C05487=1118.732,158.119,-61.971,-179.423,8.843,149.556
C05488=1118.727,158.349,-61.992,-179.422,8.846,149.556
C05489=1118.724,158.578,-62.012,-179.419,8.849,149.556
C05490=1118.719,158.807,-62.033,-179.417,8.852,149.556
C05491=1118.714,159.056,-62.056,-179.415,8.856,149.557
C05492=1118.710,159.305,-62.078,-179.412,8.859,149.557
C05493=1118.706,159.554,-62.100,-179.410,8.862,149.557
C05494=1118.701,159.803,-62.123,-179.408,8.865,149.557
C05495=1118.696,160.052,-62.145,-179.406,8.869,149.557
C05496=1118.691,160.301,-62.168,-179.403,8.872,149.557
C05497=1118.687,160.550,-62.191,-179.401,8.875,149.558
C05498=1118.683,160.799,-62.213,-179.399,8.878,149.558
C05499=1118.677,161.048,-62.236,-179.397,8.881,149.558
C05500=1118.674,161.296,-62.259,-179.394,8.884,149.558
C05501=1118.668,161.546,-62.281,-179.392,8.887,149.558
C05502=1118.664,161.794,-62.304,-179.390,8.891,149.558
C05503=1118.659,162.044,-62.326,-179.387,8.894,149.558
C05504=1118.655,162.292,-62.349,-179.385,8.898,149.558
C05505=1118.650,162.542,-62.372,-179.383,8.901,149.558
C05506=1118.645,162.790,-62.394,-179.380,8.904,149.558
C05507=1118.641,163.039,-62.417,-179.378,8.907,149.559
C05508=1118.636,163.288,-62.440,-179.376,8.910,149.559
C05509=1118.632,163.537,-62.463,-179.373,8.914,149.559
C05510=1118.627,163.785,-62.485,-179.372,8.916,149.559
C05511=1118.622,164.035,-62.508,-179.369,8.919,149.559
C05512=1118.618,164.284,-62.531,-179.367,8.923,149.559
C05513=1118.614,164.533,-62.554,-179.364,8.926,149.559
C05514=1118.609,164.781,-62.576,-179.362,8.929,149.559
C05515=1118.604,165.031,-62.599,-179.360,8.932,149.560
C05516=1118.600,165.279,-62.622,-179.357,8.936,149.560
C05517=1118.595,165.528,-62.645,-179.355,8.939,149.560
C05518=1118.591,165.777,-62.669,-179.353,8.941,149.560
C05519=1118.586,166.026,-62.690,-179.351,8.945,149.560
C05520=1118.581,166.275,-62.714,-179.348,8.948,149.560
C05521=1118.576,166.524,-62.737,-179.346,8.951,149.560
C05522=1118.572,166.773,-62.760,-179.344,8.954,149.560
C05523=1118.568,167.022,-62.783,-179.341,8.957,149.560
C05524=1118.562,167.271,-62.805,-179.340,8.960,149.560
C05525=1118.558,167.519,-62.828,-179.337,8.963,149.560
C05526=1118.553,167.768,-62.852,-179.335,8.966,149.561
C05527=1118.549,168.017,-62.875,-179.333,8.970,149.561
C05528=1118.545,168.266,-62.898,-179.330,8.973,149.561
C05529=1118.540,168.515,-62.921,-179.328,8.975,149.561
C05530=1118.535,168.764,-62.944,-179.326,8.979,149.561
C05531=1118.531,169.012,-62.967,-179.324,8.982,149.561
C05532=1118.526,169.261,-62.990,-179.321,8.985,149.561
C05533=1118.521,169.510,-63.013,-179.320,8.988,149.561
C05534=1118.517,169.759,-63.037,-179.317,8.991,149.561
C05535=1118.512,170.009,-63.059,-179.315,8.994,149.561
C05536=1118.508,170.258,-63.082,-179.312,8.997,149.561
C05537=1118.503,170.507,-63.106,-179.311,9.000,149.562
C05538=1118.498,170.755,-63.129,-179.308,9.003,149.562
C05539=1118.494,170.969,-63.149,-179.306,9.005,149.562
C05540=1118.491,171.183,-63.169,-179.304,9.009,149.562
C05541=1118.487,171.397,-63.188,-179.302,9.011,149.562
C05542=1118.482,171.610,-63.209,-179.300,9.013,149.562
C05543=1118.479,171.824,-63.229,-179.298,9.016,149.562
C05544=1118.475,172.038,-63.248,-179.297,9.018,149.562
C05545=1118.471,172.252,-63.269,-179.294,9.021,149.562
C05546=1118.467,172.466,-63.289,-179.292,9.024,149.562
C05547=1118.462,172.715,-63.312,-179.291,9.026,149.562
C05548=1118.458,172.964,-63.336,-179.289,9.029,149.563
C05549=1118.453,173.213,-63.359,-179.286,9.033,149.563
C05550=1118.449,173.461,-63.382,-179.283,9.036,149.563
C05551=1118.444,173.710,-63.405,-179.282,9.038,149.563
C05552=1118.439,173.958,-63.429,-179.279,9.042,149.563
C05553=1118.435,174.207,-63.452,-179.277,9.045,149.563
C05554=1118.430,174.456,-63.476,-179.275,9.047,149.563
C05555=1118.425,174.705,-63.499,-179.273,9.050,149.563
C05556=1118.421,174.954,-63.522,-179.270,9.054,149.563
C05557=1118.416,175.203,-63.546,-179.269,9.056,149.564
C05558=1118.412,175.451,-63.569,-179.266,9.059,149.564
C05559=1118.408,175.701,-63.592,-179.264,9.062,149.564
C05560=1118.403,175.950,-63.616,-179.262,9.065,149.564
C05561=1118.398,176.198,-63.640,-179.260,9.068,149.564
C05562=1118.394,176.447,-63.663,-179.257,9.071,149.564
C05563=1118.389,176.696,-63.687,-179.256,9.074,149.564
C05564=1118.385,176.944,-63.711,-179.253,9.077,149.564
C05565=1118.380,177.193,-63.734,-179.251,9.080,149.564
C05566=1118.375,177.442,-63.757,-179.249,9.083,149.564
C05567=1118.371,177.692,-63.782,-179.247,9.086,149.565
C05568=1118.367,177.941,-63.805,-179.244,9.089,149.565
C05569=1118.362,178.190,-63.829,-179.243,9.092,149.565
C05570=1118.358,178.438,-63.853,-179.240,9.095,149.565
C05571=1118.353,178.687,-63.876,-179.239,9.097,149.565
C05572=1118.348,178.936,-63.899,-179.236,9.100,149.565
C05573=1118.344,179.185,-63.923,-179.234,9.104,149.565
C05574=1118.339,179.434,-63.947,-179.231,9.107,149.565
C05575=1118.335,179.682,-63.971,-179.229,9.110,149.565
C05576=1118.330,179.931,-63.994,-179.226,9.113,149.565
C05577=1118.326,180.179,-64.018,-179.224,9.116,149.565
C05578=1118.321,180.428,-64.042,-179.221,9.120,149.565
C05579=1118.317,180.677,-64.066,-179.219,9.123,149.566
C05580=1118.313,180.927,-64.089,-179.215,9.126,149.565
C05581=1118.308,181.175,-64.114,-179.213,9.129,149.565
C05582=1118.303,181.424,-64.137,-179.210,9.132,149.565
C05583=1118.298,181.673,-64.162,-179.208,9.135,149.566
C05584=1118.294,181.922,-64.185,-179.205,9.139,149.566
C05585=1118.289,182.170,-64.209,-179.203,9.142,149.566
C05586=1118.285,182.419,-64.232,-179.200,9.145,149.566
C05587=1118.281,182.668,-64.257,-179.198,9.148,149.566
C05588=1118.276,182.917,-64.281,-179.195,9.151,149.566
C05589=1118.272,183.166,-64.304,-179.192,9.154,149.566
C05590=1118.266,183.415,-64.329,-179.190,9.157,149.566
C05591=1118.262,183.663,-64.353,-179.187,9.160,149.566
C05592=1118.257,183.912,-64.376,-179.184,9.163,149.566
C05593=1118.254,184.161,-64.401,-179.183,9.165,149.566
C05594=1118.249,184.410,-64.425,-179.180,9.169,149.566
C05595=1118.245,184.623,-64.445,-179.178,9.172,149.566
C05596=1118.240,184.837,-64.466,-179.176,9.174,149.566
C05597=1118.237,185.051,-64.487,-179.174,9.176,149.566
C05598=1118.233,185.264,-64.508,-179.172,9.179,149.566
C05599=1118.229,185.479,-64.528,-179.169,9.182,149.566
C05600=1118.226,185.692,-64.549,-179.167,9.184,149.566
C05601=1118.221,185.906,-64.569,-179.165,9.186,149.566
C05602=1118.218,186.120,-64.591,-179.163,9.188,149.566
C05603=1118.213,186.369,-64.614,-179.161,9.191,149.566
C05604=1118.208,186.617,-64.638,-179.158,9.195,149.566
C05605=1118.203,186.866,-64.663,-179.156,9.198,149.566
C05606=1118.200,187.115,-64.687,-179.154,9.200,149.566
C05607=1118.195,187.363,-64.711,-179.151,9.203,149.566
C05608=1118.190,187.612,-64.736,-179.149,9.206,149.566
C05609=1118.185,187.861,-64.759,-179.147,9.209,149.566
C05610=1118.182,188.110,-64.784,-179.144,9.212,149.566
C05611=1118.176,188.359,-64.809,-179.142,9.215,149.566
C05612=1118.172,188.607,-64.833,-179.140,9.217,149.566
C05613=1118.168,188.856,-64.857,-179.137,9.220,149.566
C05614=1118.163,189.105,-64.882,-179.135,9.223,149.566
C05615=1118.159,189.353,-64.906,-179.133,9.226,149.566
C05616=1118.154,189.602,-64.930,-179.130,9.229,149.566
C05617=1118.149,189.851,-64.955,-179.129,9.231,149.567
C05618=1118.145,190.100,-64.979,-179.126,9.234,149.567
C05619=1118.140,190.348,-65.004,-179.124,9.237,149.567
C05620=1118.136,190.597,-65.028,-179.122,9.240,149.567
C05621=1118.132,190.846,-65.052,-179.120,9.242,149.567
C05622=1118.127,191.095,-65.077,-179.117,9.245,149.567
C05623=1118.123,191.343,-65.101,-179.115,9.247,149.567
C05624=1118.118,191.593,-65.126,-179.114,9.250,149.567
C05625=1118.114,191.841,-65.150,-179.111,9.253,149.567
C05626=1118.108,192.090,-65.175,-179.109,9.256,149.567
C05627=1118.105,192.339,-65.199,-179.107,9.259,149.567
C05628=1118.100,192.588,-65.224,-179.105,9.261,149.567
C05629=1118.095,192.836,-65.248,-179.103,9.264,149.567
C05630=1118.091,193.085,-65.273,-179.101,9.267,149.567
C05631=1118.086,193.334,-65.297,-179.099,9.269,149.568
C05632=1118.082,193.582,-65.321,-179.097,9.272,149.568
C05633=1118.077,193.832,-65.346,-179.095,9.275,149.568
C05634=1118.073,194.079,-65.371,-179.093,9.277,149.568
C05635=1118.069,194.329,-65.396,-179.091,9.280,149.568
C05636=1118.064,194.578,-65.421,-179.089,9.283,149.568
C05637=1118.059,194.826,-65.445,-179.087,9.285,149.568
C05638=1118.055,195.075,-65.470,-179.085,9.289,149.568
C05639=1118.050,195.324,-65.494,-179.083,9.291,149.568
C05640=1118.045,195.572,-65.519,-179.081,9.294,149.568
C05641=1118.042,195.821,-65.544,-179.080,9.296,149.569
C05642=1118.037,196.070,-65.568,-179.077,9.299,149.569
C05643=1118.033,196.319,-65.593,-179.076,9.302,149.569
C05644=1118.028,196.567,-65.618,-179.073,9.305,149.569
C05645=1118.023,196.816,-65.643,-179.070,9.309,149.569
C05646=1118.019,197.065,-65.667,-179.067,9.313,149.569
C05647=1118.014,197.314,-65.692,-179.064,9.315,149.569
C05648=1118.010,197.562,-65.717,-179.061,9.319,149.569
C05649=1118.005,197.811,-65.742,-179.058,9.322,149.569
C05650=1118.001,198.060,-65.767,-179.054,9.325,149.569
C05651=1117.996,198.273,-65.788,-179.052,9.329,149.569
C05652=1117.993,198.487,-65.809,-179.049,9.331,149.569
C05653=1117.989,198.700,-65.831,-179.047,9.334,149.569
C05654=1117.985,198.914,-65.853,-179.044,9.336,149.568
C05655=1117.982,199.128,-65.874,-179.041,9.339,149.568
C05656=1117.978,199.341,-65.895,-179.038,9.342,149.568
C05657=1117.974,199.555,-65.917,-179.036,9.345,149.568
C05658=1117.970,199.768,-65.938,-179.033,9.347,149.568
C05659=1117.965,200.017,-65.964,-179.030,9.351,149.568
C05660=1117.961,200.266,-65.988,-179.027,9.354,149.568
C05661=1117.957,200.514,-66.013,-179.024,9.357,149.568
C05662=1117.952,200.763,-66.038,-179.021,9.360,149.568
C05663=1117.948,201.012,-66.063,-179.018,9.363,149.568
C05664=1117.944,201.261,-66.088,-179.015,9.366,149.568
C05665=1117.939,201.509,-66.114,-179.012,9.369,149.568
C05666=1117.934,201.759,-66.139,-179.009,9.372,149.567
C05667=1117.930,202.006,-66.163,-179.006,9.375,149.568
C05668=1117.926,202.256,-66.189,-179.003,9.378,149.567
C05669=1117.921,202.504,-66.214,-179.000,9.381,149.567
C05670=1117.917,202.753,-66.240,-178.997,9.384,149.567
C05671=1117.912,203.002,-66.265,-178.994,9.388,149.567
C05672=1117.907,203.250,-66.290,-178.991,9.390,149.567
C05673=1117.904,203.499,-66.315,-178.988,9.393,149.567
C05674=1117.899,203.747,-66.340,-178.985,9.396,149.567
C05675=1117.895,203.996,-66.366,-178.982,9.398,149.567
C05676=1117.890,204.244,-66.391,-178.980,9.402,149.567
C05677=1117.885,204.494,-66.416,-178.977,9.404,149.566
C05678=1117.881,204.743,-66.442,-178.973,9.408,149.566
C05679=1117.876,204.991,-66.467,-178.970,9.411,149.566
C05680=1117.872,205.240,-66.492,-178.968,9.414,149.566
C05681=1117.867,205.489,-66.518,-178.965,9.416,149.566
C05682=1117.863,205.737,-66.543,-178.962,9.419,149.566
C05683=1117.859,205.985,-66.569,-178.959,9.422,149.566
C05684=1117.854,206.234,-66.594,-178.957,9.425,149.566
C05685=1117.850,206.483,-66.619,-178.954,9.428,149.566
C05686=1117.845,206.732,-66.645,-178.951,9.431,149.566
C05687=1117.841,206.980,-66.670,-178.948,9.434,149.566
C05688=1117.836,207.229,-66.696,-178.945,9.436,149.566
C05689=1117.832,207.478,-66.722,-178.942,9.439,149.565
C05690=1117.827,207.726,-66.747,-178.940,9.442,149.565
C05691=1117.823,207.974,-66.773,-178.937,9.445,149.565
C05692=1117.819,208.223,-66.798,-178.934,9.448,149.565
C05693=1117.814,208.471,-66.824,-178.932,9.450,149.565
C05694=1117.810,208.721,-66.849,-178.929,9.453,149.565
C05695=1117.805,208.970,-66.875,-178.926,9.456,149.565
C05696=1117.800,209.219,-66.901,-178.924,9.459,149.565
C05697=1117.796,209.467,-66.926,-178.921,9.462,149.565
C05698=1117.791,209.716,-66.952,-178.918,9.465,149.565
C05699=1117.787,209.964,-66.978,-178.915,9.468,149.565
C05700=1117.783,210.213,-67.004,-178.913,9.471,149.565
C05701=1117.778,210.461,-67.029,-178.910,9.473,149.565
C05702=1117.774,210.710,-67.055,-178.907,9.477,149.565
C05703=1117.770,210.958,-67.081,-178.906,9.479,149.565
C05704=1117.766,211.207,-67.107,-178.903,9.482,149.565
C05705=1117.761,211.455,-67.132,-178.900,9.485,149.565
C05706=1117.756,211.704,-67.159,-178.898,9.488,149.565
C05707=1117.753,211.918,-67.181,-178.896,9.490,149.565
C05708=1117.749,212.132,-67.202,-178.893,9.493,149.565
C05709=1117.744,212.345,-67.225,-178.891,9.496,149.565
C05710=1117.741,212.558,-67.247,-178.889,9.498,149.565
C05711=1117.737,212.772,-67.270,-178.887,9.501,149.565
C05712=1117.733,212.985,-67.291,-178.885,9.503,149.565
C05713=1117.729,213.199,-67.314,-178.883,9.506,149.565
C05714=1117.726,213.412,-67.336,-178.881,9.508,149.565
C05715=1117.721,213.661,-67.362,-178.879,9.511,149.565
C05716=1117.717,213.909,-67.387,-178.877,9.514,149.565
C05717=1117.712,214.158,-67.414,-178.875,9.517,149.566
C05718=1117.708,214.407,-67.440,-178.873,9.519,149.566
C05719=1117.704,214.655,-67.466,-178.870,9.522,149.566
C05720=1117.700,214.904,-67.492,-178.868,9.525,149.566
C05721=1117.694,215.152,-67.518,-178.866,9.528,149.566
C05722=1117.690,215.401,-67.544,-178.864,9.531,149.566
C05723=1117.686,215.650,-67.570,-178.862,9.534,149.566
C05724=1117.682,215.898,-67.596,-178.860,9.537,149.566
C05725=1117.677,216.147,-67.623,-178.858,9.539,149.567
C05726=1117.673,216.396,-67.648,-178.855,9.543,149.567
C05727=1117.669,216.645,-67.674,-178.853,9.546,149.567
C05728=1117.664,216.892,-67.700,-178.851,9.548,149.567
C05729=1117.659,217.141,-67.727,-178.849,9.552,149.567
C05730=1117.655,217.389,-67.753,-178.846,9.555,149.567
C05731=1117.651,217.638,-67.779,-178.844,9.558,149.567
C05732=1117.646,217.887,-67.805,-178.842,9.560,149.567
C05733=1117.642,218.135,-67.832,-178.840,9.564,149.567
C05734=1117.638,218.384,-67.857,-178.837,9.567,149.567
C05735=1117.633,218.633,-67.884,-178.835,9.570,149.568
C05736=1117.629,218.882,-67.910,-178.833,9.573,149.568
C05737=1117.625,219.130,-67.936,-178.831,9.576,149.568
C05738=1117.620,219.378,-67.963,-178.828,9.579,149.568
C05739=1117.615,219.627,-67.988,-178.826,9.582,149.568
C05740=1117.611,219.875,-68.015,-178.824,9.585,149.568
C05741=1117.606,220.124,-68.041,-178.821,9.588,149.568
C05742=1117.602,220.372,-68.068,-178.818,9.591,149.568
C05743=1117.598,220.622,-68.094,-178.816,9.595,149.568
C05744=1117.594,220.870,-68.121,-178.813,9.598,149.569
C05745=1117.589,221.118,-68.148,-178.811,9.601,149.569
C05746=1117.585,221.367,-68.173,-178.808,9.604,149.569
C05747=1117.581,221.615,-68.200,-178.806,9.607,149.569
C05748=1117.576,221.864,-68.226,-178.803,9.610,149.569
C05749=1117.572,222.113,-68.253,-178.801,9.613,149.569
C05750=1117.567,222.361,-68.280,-178.798,9.616,149.569
C05751=1117.563,222.610,-68.305,-178.796,9.619,149.569
C05752=1117.558,222.858,-68.332,-178.793,9.623,149.569
C05753=1117.554,223.107,-68.358,-178.791,9.626,149.569
C05754=1117.550,223.356,-68.385,-178.788,9.629,149.569
C05755=1117.546,223.604,-68.412,-178.786,9.632,149.569
C05756=1117.541,223.852,-68.439,-178.783,9.635,149.569
C05757=1117.537,224.101,-68.465,-178.781,9.638,149.569
C05758=1117.532,224.350,-68.492,-178.778,9.641,149.569
C05759=1117.527,224.598,-68.519,-178.774,9.645,149.569
C05760=1117.523,224.846,-68.545,-178.772,9.648,149.569
C05761=1117.519,225.095,-68.572,-178.769,9.651,149.569
C05762=1117.515,225.344,-68.598,-178.767,9.654,149.570
C05763=1117.511,225.557,-68.621,-178.764,9.657,149.570
C05764=1117.507,225.770,-68.644,-178.762,9.659,149.569
C05765=1117.503,225.984,-68.667,-178.759,9.662,149.570
C05766=1117.500,226.197,-68.690,-178.757,9.665,149.570
C05767=1117.496,226.410,-68.713,-178.755,9.667,149.569
C05768=1117.492,226.624,-68.736,-178.752,9.670,149.570
C05769=1117.488,226.837,-68.759,-178.750,9.674,149.570
C05770=1117.484,227.051,-68.782,-178.747,9.676,149.569
C05771=1117.480,227.299,-68.808,-178.744,9.679,149.570
C05772=1117.476,227.548,-68.836,-178.741,9.682,149.569
C05773=1117.471,227.796,-68.863,-178.739,9.685,149.569
C05774=1117.467,228.045,-68.889,-178.736,9.688,149.569
C05775=1117.463,228.293,-68.916,-178.733,9.692,149.569
C05776=1117.458,228.542,-68.943,-178.730,9.695,149.569
C05777=1117.453,228.790,-68.970,-178.727,9.697,149.569
C05778=1117.449,229.038,-68.997,-178.723,9.701,149.569
C05779=1117.445,229.287,-69.024,-178.721,9.704,149.569
C05780=1117.441,229.536,-69.051,-178.717,9.708,149.569
C05781=1117.437,229.784,-69.078,-178.714,9.711,149.569
C05782=1117.432,230.033,-69.105,-178.711,9.713,149.569
C05783=1117.428,230.281,-69.132,-178.708,9.717,149.569
C05784=1117.423,230.530,-69.159,-178.705,9.720,149.569
C05785=1117.418,230.778,-69.186,-178.702,9.722,149.569
C05786=1117.415,231.027,-69.213,-178.698,9.726,149.568
C05787=1117.410,231.276,-69.240,-178.695,9.729,149.568
C05788=1117.406,231.523,-69.268,-178.693,9.732,149.568
C05789=1117.401,231.772,-69.295,-178.690,9.735,149.568
C05790=1117.397,232.020,-69.322,-178.687,9.737,149.568
C05791=1117.393,232.270,-69.349,-178.683,9.741,149.568
C05792=1117.389,232.518,-69.376,-178.681,9.744,149.568
C05793=1117.384,232.766,-69.404,-178.678,9.746,149.568
C05794=1117.380,233.014,-69.431,-178.675,9.749,149.568
C05795=1117.375,233.263,-69.458,-178.672,9.752,149.568
C05796=1117.371,233.512,-69.485,-178.669,9.755,149.568
C05797=1117.367,233.760,-69.513,-178.666,9.758,149.567
C05798=1117.362,234.008,-69.540,-178.663,9.760,149.567
C05799=1117.358,234.257,-69.567,-178.660,9.763,149.567
C05800=1117.353,234.506,-69.594,-178.657,9.766,149.567
C05801=1117.350,234.754,-69.622,-178.654,9.769,149.567
C05802=1117.345,235.002,-69.649,-178.652,9.771,149.567
C05803=1117.341,235.251,-69.677,-178.649,9.775,149.567
C05804=1117.337,235.499,-69.704,-178.647,9.777,149.567
C05805=1117.332,235.748,-69.731,-178.644,9.779,149.567
C05806=1117.327,235.995,-69.759,-178.641,9.782,149.567
C05807=1117.323,236.245,-69.786,-178.638,9.785,149.566
C05808=1117.319,236.493,-69.813,-178.635,9.788,149.566
C05809=1117.314,236.741,-69.841,-178.633,9.789,149.566
C05810=1117.310,236.990,-69.868,-178.630,9.793,149.566
C05811=1117.306,237.238,-69.896,-178.627,9.795,149.566
C05812=1117.301,237.487,-69.923,-178.624,9.798,149.566
C05813=1117.298,237.735,-69.951,-178.622,9.800,149.566
C05814=1117.293,237.984,-69.978,-178.619,9.803,149.566
C05815=1117.289,238.232,-70.006,-178.616,9.806,149.566
C05816=1117.284,238.481,-70.034,-178.614,9.808,149.566
C05817=1117.279,238.729,-70.062,-178.611,9.811,149.566
C05818=1117.275,238.977,-70.089,-178.609,9.813,149.566
C05819=1117.272,239.191,-70.113,-178.606,9.816,149.565
C05820=1117.268,239.404,-70.137,-178.604,9.818,149.565
C05821=1117.264,239.617,-70.160,-178.602,9.820,149.565
C05822=1117.261,239.830,-70.184,-178.600,9.822,149.565
C05823=1117.257,240.044,-70.209,-178.598,9.824,149.565
C05824=1117.253,240.257,-70.232,-178.596,9.826,149.565
C05825=1117.249,240.470,-70.256,-178.594,9.829,149.565
C05826=1117.246,240.683,-70.279,-178.591,9.831,149.565
C05827=1117.242,240.931,-70.307,-178.589,9.833,149.565
C05828=1117.237,241.180,-70.335,-178.586,9.836,149.565
C05829=1117.233,241.429,-70.363,-178.584,9.838,149.565
C05830=1117.228,241.677,-70.391,-178.582,9.841,149.565
C05831=1117.224,241.926,-70.418,-178.579,9.843,149.565
C05832=1117.220,242.174,-70.446,-178.577,9.845,149.565
C05833=1117.216,242.421,-70.474,-178.575,9.848,149.565
C05834=1117.211,242.671,-70.502,-178.573,9.850,149.565
C05835=1117.207,242.919,-70.530,-178.570,9.853,149.565
C05836=1117.203,243.167,-70.558,-178.568,9.855,149.565
C05837=1117.198,243.415,-70.586,-178.566,9.858,149.565
C05838=1117.194,243.665,-70.613,-178.563,9.861,149.565
C05839=1117.189,243.913,-70.641,-178.561,9.863,149.565
C05840=1117.185,244.161,-70.669,-178.559,9.865,149.565
C05841=1117.181,244.409,-70.697,-178.557,9.867,149.565
C05842=1117.177,244.657,-70.725,-178.555,9.870,149.565
C05843=1117.172,244.907,-70.753,-178.553,9.873,149.565
C05844=1117.168,245.154,-70.781,-178.551,9.875,149.565
C05845=1117.164,245.403,-70.809,-178.549,9.877,149.565
C05846=1117.160,245.651,-70.837,-178.546,9.880,149.565
C05847=1117.155,245.900,-70.866,-178.544,9.883,149.565
C05848=1117.151,246.148,-70.893,-178.542,9.885,149.565
C05849=1117.147,246.396,-70.922,-178.540,9.887,149.565
C05850=1117.142,246.645,-70.949,-178.538,9.890,149.565
C05851=1117.138,246.894,-70.977,-178.536,9.893,149.566
C05852=1117.134,247.141,-71.005,-178.535,9.895,149.566
C05853=1117.129,247.390,-71.034,-178.533,9.898,149.566
C05854=1117.125,247.638,-71.062,-178.529,9.901,149.566
C05855=1117.121,247.887,-71.090,-178.524,9.905,149.565
C05856=1117.116,248.135,-71.118,-178.520,9.909,149.565
C05857=1117.112,248.384,-71.146,-178.515,9.913,149.565
C05858=1117.108,248.631,-71.174,-178.511,9.917,149.564
C05859=1117.103,248.880,-71.203,-178.507,9.920,149.564
C05860=1117.100,249.129,-71.231,-178.502,9.925,149.564
C05861=1117.094,249.377,-71.259,-178.498,9.928,149.564
C05862=1117.091,249.626,-71.287,-178.494,9.931,149.564
C05863=1117.086,249.873,-71.317,-178.490,9.934,149.563
C05864=1117.082,250.122,-71.345,-178.486,9.937,149.563
C05865=1117.078,250.370,-71.372,-178.482,9.940,149.563
C05866=1117.073,250.619,-71.401,-178.479,9.944,149.563
C05867=1117.070,250.867,-71.429,-178.475,9.946,149.562
C05868=1117.064,251.115,-71.458,-178.472,9.949,149.562
C05869=1117.061,251.363,-71.487,-178.469,9.952,149.562
C05870=1117.057,251.612,-71.515,-178.465,9.955,149.562
C05871=1117.052,251.860,-71.543,-178.462,9.957,149.561
C05872=1117.048,252.109,-71.572,-178.460,9.959,149.561
C05873=1117.044,252.357,-71.601,-178.457,9.962,149.561
C05874=1117.039,252.605,-71.629,-178.454,9.965,149.561
C05875=1117.036,252.819,-71.654,-178.451,9.966,149.561
C05876=1117.032,253.032,-71.678,-178.449,9.969,149.561
C05877=1117.028,253.245,-71.703,-178.448,9.970,149.561
C05878=1117.025,253.457,-71.727,-178.445,9.972,149.561
C05879=1117.021,253.671,-71.752,-178.443,9.974,149.560
C05880=1117.017,253.884,-71.776,-178.442,9.976,149.560
C05881=1117.014,254.097,-71.801,-178.440,9.977,149.560
C05882=1117.010,254.310,-71.826,-178.438,9.979,149.560
C05883=1117.005,254.559,-71.855,-178.436,9.981,149.560
C05884=1117.001,254.807,-71.882,-178.435,9.983,149.560
C05885=1116.997,255.055,-71.912,-178.433,9.985,149.560
C05886=1116.993,255.304,-71.940,-178.432,9.986,149.560
C05887=1116.989,255.552,-71.969,-178.431,9.988,149.561
C05888=1116.984,255.800,-71.998,-178.429,9.990,149.561
C05889=1116.980,256.049,-72.026,-178.428,9.992,149.561
C05890=1116.976,256.297,-72.055,-178.425,9.995,149.561
C05891=1116.971,256.545,-72.084,-178.422,9.998,149.561
C05892=1116.967,256.793,-72.113,-178.419,10.001,149.561
C05893=1116.963,257.042,-72.141,-178.417,10.003,149.560
C05894=1116.959,257.290,-72.171,-178.414,10.006,149.561
C05895=1116.954,257.538,-72.199,-178.411,10.009,149.560
C05896=1116.950,257.786,-72.228,-178.408,10.012,149.560
C05897=1116.946,258.035,-72.257,-178.405,10.014,149.560
C05898=1116.942,258.282,-72.285,-178.403,10.017,149.560
C05899=1116.937,258.531,-72.314,-178.400,10.020,149.560
C05900=1116.933,258.780,-72.343,-178.397,10.023,149.560
C05901=1116.928,259.028,-72.372,-178.394,10.026,149.560
C05902=1116.925,259.276,-72.401,-178.391,10.029,149.560
C05903=1116.920,259.524,-72.430,-178.388,10.032,149.560
C05904=1116.916,259.773,-72.459,-178.385,10.035,149.560
C05905=1116.912,260.021,-72.488,-178.382,10.037,149.560
C05906=1116.908,260.269,-72.517,-178.379,10.040,149.559
C05907=1116.904,260.518,-72.546,-178.376,10.043,149.559
C05908=1116.899,260.766,-72.575,-178.373,10.046,149.559
C05909=1116.895,261.014,-72.604,-178.370,10.048,149.559
C05910=1116.890,261.263,-72.633,-178.367,10.051,149.559
C05911=1116.887,261.511,-72.662,-178.363,10.054,149.559
C05912=1116.883,261.759,-72.691,-178.360,10.057,149.559
C05913=1116.878,262.006,-72.721,-178.357,10.060,149.559
C05914=1116.873,262.255,-72.749,-178.354,10.063,149.558
C05915=1116.869,262.504,-72.779,-178.351,10.065,149.558
C05916=1116.865,262.752,-72.808,-178.347,10.069,149.558
C05917=1116.861,263.000,-72.838,-178.344,10.071,149.558
C05918=1116.856,263.249,-72.866,-178.341,10.074,149.558
C05919=1116.852,263.497,-72.896,-178.338,10.077,149.558
C05920=1116.848,263.745,-72.924,-178.334,10.080,149.557
C05921=1116.844,263.993,-72.954,-178.332,10.083,149.557
C05922=1116.840,264.241,-72.983,-178.328,10.085,149.557
C05923=1116.836,264.489,-73.013,-178.325,10.088,149.557
C05924=1116.831,264.738,-73.042,-178.322,10.091,149.557
C05925=1116.827,264.986,-73.072,-178.319,10.094,149.557
C05926=1116.823,265.234,-73.101,-178.317,10.095,149.557
C05927=1116.819,265.482,-73.131,-178.314,10.098,149.556
C05928=1116.814,265.731,-73.159,-178.312,10.100,149.556
C05929=1116.810,265.980,-73.189,-178.309,10.103,149.556
C05930=1116.805,266.227,-73.218,-178.306,10.106,149.556
C05931=1116.802,266.440,-73.244,-178.304,10.108,149.556
C05932=1116.799,266.653,-73.269,-178.301,10.110,149.556
C05933=1116.794,266.866,-73.294,-178.299,10.112,149.556
C05934=1116.791,267.079,-73.320,-178.297,10.114,149.556
C05935=1116.788,267.292,-73.345,-178.294,10.116,149.556
C05936=1116.784,267.506,-73.370,-178.292,10.118,149.555
C05937=1116.780,267.718,-73.395,-178.290,10.121,149.556
C05938=1116.777,267.931,-73.421,-178.287,10.123,149.555
C05939=1116.772,268.179,-73.450,-178.284,10.125,149.555
C05940=1116.768,268.428,-73.480,-178.282,10.127,149.555
C05941=1116.764,268.676,-73.509,-178.279,10.130,149.555
C05942=1116.760,268.924,-73.539,-178.276,10.133,149.555
C05943=1116.755,269.172,-73.569,-178.274,10.135,149.555
C05944=1116.751,269.421,-73.599,-178.271,10.138,149.555
C05945=1116.747,269.669,-73.628,-178.268,10.140,149.555
C05946=1116.743,269.917,-73.658,-178.265,10.143,149.555
C05947=1116.738,270.165,-73.687,-178.262,10.146,149.554
C05948=1116.735,270.413,-73.717,-178.260,10.148,149.554
C05949=1116.730,270.661,-73.747,-178.257,10.151,149.554
C05950=1116.726,270.909,-73.776,-178.254,10.154,149.554
C05951=1116.721,271.158,-73.806,-178.251,10.156,149.554
C05952=1116.717,271.406,-73.836,-178.248,10.159,149.554
C05953=1116.713,271.654,-73.866,-178.245,10.161,149.554
C05954=1116.709,271.902,-73.895,-178.242,10.163,149.553
C05955=1116.705,272.151,-73.925,-178.239,10.166,149.553
C05956=1116.700,272.398,-73.955,-178.237,10.169,149.553
C05957=1116.696,272.647,-73.985,-178.234,10.172,149.553
C05958=1116.692,272.895,-74.014,-178.231,10.174,149.553
C05959=1116.688,273.143,-74.045,-178.228,10.177,149.553
C05960=1116.684,273.391,-74.074,-178.225,10.179,149.553
C05961=1116.680,273.640,-74.105,-178.222,10.182,149.553
C05962=1116.676,273.888,-74.135,-178.220,10.185,149.553
C05963=1116.671,274.136,-74.164,-178.216,10.187,149.552
C05964=1116.667,274.384,-74.195,-178.213,10.190,149.552
C05965=1116.663,274.632,-74.224,-178.210,10.193,149.552
C05966=1116.659,274.880,-74.254,-178.207,10.195,149.552
C05967=1116.655,275.128,-74.284,-178.204,10.198,149.552
C05968=1116.650,275.376,-74.315,-178.201,10.201,149.552
C05969=1116.646,275.624,-74.344,-178.199,10.204,149.552
C05970=1116.643,275.873,-74.375,-178.195,10.206,149.552
C05971=1116.638,276.121,-74.405,-178.192,10.209,149.551
C05972=1116.634,276.369,-74.435,-178.189,10.212,149.551
C05973=1116.630,276.617,-74.464,-178.186,10.214,149.551
C05974=1116.625,276.865,-74.495,-178.183,10.217,149.551
C05975=1116.621,277.114,-74.524,-178.180,10.220,149.551
C05976=1116.618,277.362,-74.555,-178.177,10.222,149.551
C05977=1116.613,277.610,-74.586,-178.174,10.225,149.551
C05978=1116.609,277.858,-74.615,-178.171,10.228,149.550
C05979=1116.604,278.106,-74.646,-178.168,10.230,149.550
C05980=1116.600,278.354,-74.676,-178.165,10.233,149.550
C05981=1116.597,278.603,-74.706,-178.162,10.235,149.550
C05982=1116.592,278.851,-74.737,-178.159,10.238,149.550
C05983=1116.588,279.098,-74.767,-178.155,10.241,149.550
C05984=1116.583,279.347,-74.797,-178.152,10.243,149.549
C05985=1116.579,279.595,-74.827,-178.150,10.246,149.549
C05986=1116.575,279.843,-74.858,-178.146,10.249,149.549
C05987=1116.571,280.055,-74.884,-178.143,10.251,149.549
C05988=1116.568,280.268,-74.910,-178.141,10.253,149.549
C05989=1116.564,280.481,-74.936,-178.138,10.256,149.549
C05990=1116.561,280.694,-74.962,-178.135,10.258,149.548
C05991=1116.557,280.907,-74.989,-178.132,10.261,149.548
C05992=1116.554,281.120,-75.014,-178.130,10.262,149.548
C05993=1116.550,281.333,-75.040,-178.127,10.265,149.548
C05994=1116.546,281.546,-75.067,-178.124,10.267,149.548
C05995=1116.543,281.793,-75.097,-178.121,10.270,149.548
C05996=1116.538,282.042,-75.127,-178.118,10.272,149.547
C05997=1116.534,282.290,-75.158,-178.115,10.275,149.547
C05998=1116.530,282.538,-75.188,-178.112,10.277,149.547
C05999=1116.525,282.786,-75.219,-178.109,10.280,149.547
C06000=1116.521,283.034,-75.249,-178.107,10.282,149.547
C06001=1116.517,283.283,-75.280,-178.103,10.284,149.547
C06002=1116.513,283.531,-75.311,-178.100,10.287,149.546
C06003=1116.509,283.778,-75.341,-178.097,10.290,149.546
C06004=1116.505,284.027,-75.373,-178.094,10.292,149.546
C06005=1116.501,284.274,-75.403,-178.091,10.295,149.546
C06006=1116.496,284.522,-75.433,-178.088,10.298,149.546
C06007=1116.492,284.771,-75.465,-178.085,10.300,149.546
C06008=1116.488,285.019,-75.495,-178.081,10.303,149.545
C06009=1116.484,285.267,-75.526,-178.079,10.305,149.545
C06010=1116.480,285.515,-75.557,-178.076,10.307,149.545
C06011=1116.476,285.763,-75.587,-178.073,10.310,149.545
C06012=1116.471,286.011,-75.618,-178.070,10.312,149.545
C06013=1116.467,286.260,-75.649,-178.067,10.315,149.545
C06014=1116.463,286.508,-75.679,-178.064,10.318,149.544
C06015=1116.459,286.755,-75.710,-178.060,10.320,149.544
C06016=1116.455,287.003,-75.741,-178.057,10.323,149.544
C06017=1116.450,287.251,-75.772,-178.054,10.325,149.544
C06018=1116.447,287.500,-75.803,-178.052,10.327,149.544
C06019=1116.443,287.748,-75.834,-178.048,10.330,149.543
C06020=1116.438,287.995,-75.864,-178.046,10.333,149.543
C06021=1116.434,288.244,-75.895,-178.043,10.335,149.543
C06022=1116.430,288.491,-75.927,-178.039,10.338,149.543
C06023=1116.426,288.740,-75.957,-178.036,10.341,149.543
C06024=1116.422,288.988,-75.988,-178.033,10.343,149.543
C06025=1116.418,289.236,-76.019,-178.030,10.346,149.542
C06026=1116.413,289.484,-76.051,-178.027,10.348,149.542
C06027=1116.409,289.732,-76.082,-178.024,10.350,149.542
C06028=1116.406,289.980,-76.112,-178.021,10.353,149.542
C06029=1116.401,290.227,-76.144,-178.018,10.355,149.542
C06030=1116.397,290.476,-76.175,-178.015,10.358,149.542
C06031=1116.393,290.724,-76.205,-178.012,10.361,149.541
C06032=1116.389,290.972,-76.237,-178.009,10.363,149.541
C06033=1116.384,291.220,-76.268,-178.006,10.366,149.541
C06034=1116.380,291.469,-76.299,-178.003,10.368,149.541
C06035=1116.377,291.716,-76.330,-177.999,10.371,149.541
C06036=1116.373,291.964,-76.361,-177.997,10.373,149.541
C06037=1116.368,292.212,-76.393,-177.994,10.375,149.540
C06038=1116.364,292.460,-76.424,-177.991,10.378,149.540
C06039=1116.360,292.708,-76.455,-177.987,10.381,149.540
C06040=1116.356,292.956,-76.486,-177.984,10.383,149.540
C06041=1116.352,293.204,-76.518,-177.981,10.386,149.540
C06042=1116.348,293.452,-76.549,-177.978,10.388,149.539
C06043=1116.344,293.665,-76.576,-177.976,10.390,149.539
C06044=1116.341,293.878,-76.602,-177.973,10.393,149.539
C06045=1116.337,294.090,-76.629,-177.970,10.395,149.539
C06046=1116.333,294.303,-76.657,-177.968,10.397,149.539
C06047=1116.329,294.516,-76.683,-177.965,10.400,149.539
C06048=1116.327,294.729,-76.710,-177.962,10.401,149.538
C06049=1116.323,294.941,-76.737,-177.960,10.403,149.538
C06050=1116.320,295.154,-76.764,-177.957,10.406,149.538
C06051=1116.315,295.402,-76.795,-177.954,10.408,149.538
C06052=1116.311,295.650,-76.827,-177.951,10.410,149.538
C06053=1116.307,295.898,-76.858,-177.949,10.413,149.538
C06054=1116.303,296.146,-76.890,-177.945,10.416,149.538
C06055=1116.299,296.394,-76.922,-177.942,10.418,149.537
C06056=1116.295,296.642,-76.952,-177.939,10.421,149.537
C06057=1116.291,296.890,-76.984,-177.936,10.424,149.537
C06058=1116.287,297.138,-77.016,-177.933,10.426,149.537
C06059=1116.282,297.385,-77.048,-177.930,10.429,149.537
C06060=1116.278,297.634,-77.079,-177.926,10.431,149.536
C06061=1116.274,297.881,-77.111,-177.924,10.433,149.536
C06062=1116.270,298.129,-77.143,-177.921,10.436,149.536
C06063=1116.267,298.377,-77.174,-177.918,10.438,149.536
C06064=1116.262,298.625,-77.205,-177.914,10.441,149.536
C06065=1116.258,298.873,-77.237,-177.912,10.444,149.536
C06066=1116.253,299.121,-77.269,-177.908,10.446,149.535
C06067=1116.249,299.369,-77.301,-177.905,10.449,149.535
C06068=1116.246,299.617,-77.333,-177.902,10.451,149.535
C06069=1116.241,299.864,-77.364,-177.899,10.454,149.535
C06070=1116.237,300.113,-77.395,-177.896,10.456,149.535
C06071=1116.234,300.361,-77.427,-177.893,10.458,149.535
C06072=1116.229,300.609,-77.459,-177.890,10.461,149.534
C06073=1116.225,300.857,-77.491,-177.887,10.464,149.534
C06074=1116.221,301.105,-77.523,-177.884,10.466,149.534
C06075=1116.217,301.352,-77.554,-177.881,10.469,149.534
C06076=1116.213,301.601,-77.587,-177.877,10.471,149.534
C06077=1116.209,301.849,-77.619,-177.875,10.474,149.534
C06078=1116.205,302.096,-77.650,-177.871,10.476,149.533
C06079=1116.200,302.344,-77.683,-177.868,10.479,149.533
C06080=1116.196,302.592,-77.714,-177.865,10.482,149.533
C06081=1116.193,302.840,-77.746,-177.863,10.484,149.533
C06082=1116.188,303.088,-77.778,-177.859,10.486,149.533
C06083=1116.184,303.336,-77.810,-177.856,10.489,149.533
C06084=1116.180,303.584,-77.842,-177.853,10.491,149.532
C06085=1116.176,303.832,-77.875,-177.850,10.494,149.532
C06086=1116.171,304.080,-77.906,-177.847,10.497,149.532
C06087=1116.168,304.328,-77.938,-177.843,10.499,149.532
C06088=1116.163,304.576,-77.970,-177.841,10.502,149.532
C06089=1116.159,304.823,-78.003,-177.837,10.504,149.531
C06090=1116.156,305.071,-78.034,-177.834,10.507,149.531
C06091=1116.151,305.319,-78.067,-177.832,10.509,149.531
C06092=1116.147,305.567,-78.099,-177.829,10.511,149.531
C06093=1116.143,305.816,-78.131,-177.825,10.514,149.531
C06094=1116.139,306.063,-78.163,-177.822,10.517,149.531
C06095=1116.135,306.310,-78.195,-177.819,10.519,149.530
C06096=1116.131,306.559,-78.228,-177.816,10.522,149.530
C06097=1116.127,306.807,-78.259,-177.813,10.524,149.530
C06098=1116.123,307.055,-78.292,-177.810,10.527,149.530
C06099=1116.119,307.267,-78.320,-177.807,10.529,149.530
C06100=1116.116,307.479,-78.347,-177.804,10.531,149.529
C06101=1116.113,307.693,-78.375,-177.802,10.533,149.529
C06102=1116.109,307.905,-78.402,-177.799,10.535,149.529
C06103=1116.105,308.117,-78.430,-177.796,10.538,149.529
C06104=1116.102,308.330,-78.459,-177.794,10.540,149.529
C06105=1116.098,308.542,-78.486,-177.791,10.541,149.529
C06106=1116.095,308.755,-78.513,-177.788,10.544,149.529
C06107=1116.090,309.003,-78.546,-177.785,10.547,149.528
C06108=1116.087,309.251,-78.578,-177.783,10.549,149.528
C06109=1116.083,309.498,-78.611,-177.779,10.551,149.528
C06110=1116.079,309.746,-78.643,-177.777,10.554,149.528
C06111=1116.074,309.995,-78.675,-177.773,10.556,149.528
C06112=1116.071,310.242,-78.708,-177.770,10.559,149.528
C06113=1116.066,310.490,-78.740,-177.767,10.562,149.527
C06114=1116.063,310.737,-78.773,-177.764,10.564,149.527
C06115=1116.058,310.986,-78.805,-177.761,10.567,149.527
C06116=1116.054,311.233,-78.838,-177.757,10.569,149.527
C06117=1116.050,311.481,-78.870,-177.754,10.572,149.527
C06118=1116.046,311.729,-78.903,-177.751,10.574,149.526
C06119=1116.042,311.977,-78.935,-177.749,10.576,149.526
C06120=1116.038,312.225,-78.968,-177.745,10.579,149.526
C06121=1116.034,312.473,-79.001,-177.743,10.582,149.526
C06122=1116.030,312.721,-79.033,-177.739,10.584,149.526
C06123=1116.026,312.968,-79.066,-177.736,10.586,149.525
C06124=1116.022,313.217,-79.099,-177.733,10.589,149.525
C06125=1116.019,313.464,-79.131,-177.730,10.592,149.525
C06126=1116.014,313.711,-79.164,-177.727,10.594,149.525
C06127=1116.009,313.959,-79.197,-177.723,10.597,149.525
C06128=1116.006,314.207,-79.229,-177.720,10.600,149.525
C06129=1116.002,314.455,-79.262,-177.717,10.602,149.524
C06130=1115.997,314.703,-79.295,-177.714,10.604,149.524
C06131=1115.994,314.950,-79.327,-177.711,10.607,149.524
C06132=1115.990,315.198,-79.360,-177.708,10.609,149.524
C06133=1115.985,315.446,-79.393,-177.705,10.612,149.524
C06134=1115.981,315.694,-79.426,-177.702,10.614,149.524
C06135=1115.978,315.942,-79.459,-177.699,10.617,149.523
C06136=1115.974,316.189,-79.492,-177.696,10.619,149.523
C06137=1115.970,316.437,-79.525,-177.692,10.622,149.523
C06138=1115.965,316.685,-79.557,-177.689,10.625,149.523
C06139=1115.962,316.933,-79.590,-177.686,10.627,149.523
C06140=1115.958,317.181,-79.623,-177.683,10.629,149.522
C06141=1115.954,317.429,-79.657,-177.680,10.631,149.522
C06142=1115.950,317.677,-79.690,-177.677,10.634,149.522
C06143=1115.946,317.924,-79.723,-177.674,10.637,149.522
C06144=1115.942,318.172,-79.755,-177.671,10.639,149.522
C06145=1115.938,318.420,-79.788,-177.668,10.642,149.521
C06146=1115.934,318.668,-79.821,-177.665,10.644,149.521
C06147=1115.930,318.916,-79.854,-177.661,10.647,149.521
C06148=1115.926,319.163,-79.887,-177.658,10.649,149.521
C06149=1115.921,319.411,-79.921,-177.655,10.652,149.521
C06150=1115.917,319.659,-79.954,-177.652,10.654,149.521
C06151=1115.914,319.906,-79.986,-177.649,10.657,149.520
C06152=1115.910,320.154,-80.019,-177.646,10.659,149.520
C06153=1115.906,320.402,-80.053,-177.643,10.661,149.520
C06154=1115.902,320.650,-80.086,-177.640,10.664,149.520
C06155=1115.898,320.862,-80.115,-177.637,10.667,149.520
C06156=1115.895,321.075,-80.143,-177.634,10.669,149.520
C06157=1115.891,321.287,-80.171,-177.632,10.671,149.519
C06158=1115.889,321.499,-80.200,-177.629,10.673,149.519
C06159=1115.885,321.712,-80.229,-177.626,10.675,149.519
C06160=1115.882,321.924,-80.257,-177.624,10.677,149.519
C06161=1115.878,322.137,-80.286,-177.621,10.679,149.519
C06162=1115.875,322.349,-80.314,-177.618,10.681,149.519
C06163=1115.871,322.597,-80.348,-177.615,10.684,149.518
C06164=1115.867,322.845,-80.381,-177.612,10.686,149.518
C06165=1115.863,323.092,-80.414,-177.609,10.689,149.518
C06166=1115.859,323.340,-80.448,-177.606,10.692,149.518
C06167=1115.855,323.587,-80.481,-177.602,10.694,149.518
C06168=1115.851,323.835,-80.514,-177.599,10.697,149.518
C06169=1115.847,324.083,-80.548,-177.596,10.699,149.517
C06170=1115.843,324.331,-80.581,-177.593,10.701,149.517
C06171=1115.839,324.579,-80.615,-177.590,10.704,149.517
C06172=1115.834,324.826,-80.648,-177.587,10.706,149.517
C06173=1115.830,325.074,-80.682,-177.584,10.709,149.516
C06174=1115.827,325.322,-80.716,-177.581,10.711,149.516
C06175=1115.823,325.570,-80.749,-177.577,10.714,149.516
C06176=1115.819,325.817,-80.782,-177.574,10.716,149.516
C06177=1115.815,326.064,-80.816,-177.571,10.719,149.516
C06178=1115.811,326.312,-80.849,-177.568,10.721,149.516
C06179=1115.807,326.561,-80.883,-177.565,10.724,149.515
C06180=1115.803,326.808,-80.916,-177.562,10.727,149.515
C06181=1115.799,327.056,-80.950,-177.559,10.728,149.515
C06182=1115.795,327.303,-80.984,-177.556,10.731,149.515
C06183=1115.791,327.551,-81.018,-177.553,10.734,149.515
C06184=1115.787,327.799,-81.051,-177.549,10.736,149.514
C06185=1115.783,328.046,-81.085,-177.546,10.738,149.514
C06186=1115.779,328.294,-81.118,-177.543,10.741,149.514
C06187=1115.775,328.542,-81.153,-177.540,10.744,149.514
C06188=1115.771,328.790,-81.186,-177.537,10.746,149.514
C06189=1115.767,329.037,-81.220,-177.534,10.749,149.514
C06190=1115.764,329.285,-81.253,-177.530,10.751,149.513
C06191=1115.759,329.533,-81.288,-177.527,10.754,149.513
C06192=1115.755,329.780,-81.322,-177.524,10.757,149.513
C06193=1115.752,330.028,-81.355,-177.521,10.758,149.513
C06194=1115.748,330.275,-81.389,-177.518,10.761,149.513
C06195=1115.743,330.523,-81.423,-177.515,10.763,149.512
C06196=1115.739,330.770,-81.457,-177.512,10.766,149.512
C06197=1115.736,331.018,-81.491,-177.508,10.768,149.512
C06198=1115.731,331.266,-81.525,-177.505,10.771,149.512
C06199=1115.727,331.513,-81.558,-177.502,10.774,149.512
C06200=1115.724,331.761,-81.593,-177.499,10.776,149.512
C06201=1115.720,332.009,-81.626,-177.496,10.779,149.511
C06202=1115.716,332.257,-81.661,-177.492,10.781,149.511
C06203=1115.712,332.504,-81.695,-177.489,10.784,149.511
C06204=1115.708,332.752,-81.728,-177.486,10.786,149.511
C06205=1115.704,333.000,-81.763,-177.483,10.788,149.510
C06206=1115.700,333.247,-81.796,-177.480,10.791,149.510
C06207=1115.695,333.495,-81.831,-177.477,10.793,149.510
C06208=1115.692,333.743,-81.864,-177.474,10.796,149.510
C06209=1115.688,333.990,-81.898,-177.470,10.798,149.510
C06210=1115.684,334.238,-81.933,-177.468,10.801,149.510
C06211=1115.680,334.450,-81.962,-177.465,10.803,149.509
C06212=1115.677,334.662,-81.992,-177.462,10.805,149.509
C06213=1115.674,334.875,-82.021,-177.459,10.807,149.509
C06214=1115.671,335.087,-82.050,-177.457,10.809,149.509
C06215=1115.668,335.299,-82.079,-177.454,10.811,149.509
C06216=1115.664,335.511,-82.109,-177.451,10.813,149.509
C06217=1115.661,335.723,-82.137,-177.448,10.816,149.508
C06218=1115.657,335.936,-82.167,-177.446,10.818,149.508
C06219=1115.653,336.184,-82.202,-177.442,10.820,149.508
C06220=1115.650,336.431,-82.236,-177.439,10.823,149.508
C06221=1115.645,336.678,-82.270,-177.436,10.826,149.508
C06222=1115.642,336.926,-82.305,-177.433,10.828,149.508
C06223=1115.637,337.174,-82.339,-177.430,10.830,149.507
C06224=1115.634,337.421,-82.373,-177.427,10.832,149.507
C06225=1115.629,337.669,-82.408,-177.424,10.835,149.507
C06226=1115.626,337.917,-82.442,-177.421,10.837,149.507
C06227=1115.622,338.164,-82.476,-177.417,10.840,149.507
C06228=1115.618,338.412,-82.511,-177.414,10.842,149.506
C06229=1115.614,338.659,-82.545,-177.411,10.845,149.506
C06230=1115.610,338.907,-82.580,-177.408,10.848,149.506
C06231=1115.606,339.155,-82.614,-177.404,10.850,149.506
C06232=1115.602,339.403,-82.649,-177.401,10.852,149.506
C06233=1115.598,339.650,-82.682,-177.398,10.855,149.505
C06234=1115.595,339.897,-82.718,-177.395,10.858,149.505
C06235=1115.590,340.145,-82.753,-177.392,10.859,149.505
C06236=1115.587,340.392,-82.787,-177.389,10.862,149.505
C06237=1115.582,340.640,-82.821,-177.386,10.864,149.505
C06238=1115.578,340.888,-82.856,-177.383,10.867,149.504
C06239=1115.575,341.135,-82.891,-177.379,10.870,149.504
C06240=1115.571,341.383,-82.925,-177.376,10.872,149.504
C06241=1115.566,341.630,-82.960,-177.373,10.874,149.504
C06242=1115.563,341.878,-82.994,-177.369,10.877,149.504
C06243=1115.559,342.125,-83.030,-177.366,10.880,149.503
C06244=1115.555,342.373,-83.064,-177.363,10.882,149.503
C06245=1115.551,342.621,-83.098,-177.360,10.885,149.503
C06246=1115.547,342.868,-83.133,-177.357,10.887,149.503
C06247=1115.543,343.116,-83.168,-177.354,10.889,149.503
C06248=1115.539,343.363,-83.203,-177.351,10.892,149.502
C06249=1115.535,343.611,-83.237,-177.348,10.894,149.502
C06250=1115.532,343.858,-83.273,-177.344,10.896,149.502
C06251=1115.527,344.106,-83.307,-177.341,10.899,149.502
C06252=1115.524,344.353,-83.343,-177.338,10.901,149.502
C06253=1115.520,344.600,-83.377,-177.335,10.904,149.502
C06254=1115.516,344.848,-83.411,-177.331,10.907,149.501
C06255=1115.512,345.096,-83.447,-177.328,10.909,149.501
C06256=1115.507,345.343,-83.481,-177.325,10.912,149.501
C06257=1115.504,345.591,-83.517,-177.322,10.914,149.501
C06258=1115.501,345.839,-83.551,-177.319,10.916,149.500
C06259=1115.496,346.085,-83.586,-177.316,10.918,149.500
C06260=1115.492,346.334,-83.621,-177.313,10.921,149.500
C06261=1115.489,346.581,-83.657,-177.309,10.923,149.500
C06262=1115.484,346.828,-83.691,-177.306,10.926,149.500
C06263=1115.480,347.076,-83.727,-177.303,10.928,149.499
C06264=1115.477,347.323,-83.762,-177.299,10.931,149.499
C06265=1115.473,347.571,-83.796,-177.296,10.934,149.499
C06266=1115.469,347.818,-83.832,-177.293,10.936,149.499
C06267=1115.465,348.031,-83.862,-177.290,10.938,149.499
C06268=1115.462,348.243,-83.892,-177.288,10.940,149.499
C06269=1115.459,348.455,-83.922,-177.285,10.942,149.498
C06270=1115.455,348.667,-83.952,-177.282,10.944,149.498
C06271=1115.452,348.879,-83.982,-177.279,10.947,149.498
C06272=1115.449,349.091,-84.012,-177.277,10.948,149.498
C06273=1115.446,349.303,-84.043,-177.274,10.950,149.498
C06274=1115.442,349.515,-84.072,-177.271,10.953,149.497
C06275=1115.439,349.763,-84.108,-177.268,10.955,149.497
C06276=1115.435,350.010,-84.144,-177.264,10.958,149.497
C06277=1115.430,350.258,-84.178,-177.261,10.960,149.497
C06278=1115.427,350.505,-84.214,-177.258,10.963,149.497
C06279=1115.423,350.753,-84.249,-177.254,10.965,149.496
C06280=1115.419,351.000,-84.285,-177.251,10.968,149.496
C06281=1115.415,351.248,-84.319,-177.248,10.970,149.496
C06282=1115.411,351.495,-84.355,-177.244,10.973,149.496
C06283=1115.408,351.743,-84.390,-177.241,10.976,149.495
C06284=1115.404,351.990,-84.426,-177.237,10.978,149.495
C06285=1115.400,352.238,-84.461,-177.234,10.980,149.495
C06286=1115.396,352.484,-84.497,-177.230,10.983,149.495
C06287=1115.392,352.732,-84.532,-177.227,10.985,149.494
C06288=1115.389,352.979,-84.568,-177.224,10.988,149.494
C06289=1115.385,353.227,-84.602,-177.220,10.990,149.494
C06290=1115.381,353.475,-84.638,-177.217,10.993,149.494
C06291=1115.377,353.723,-84.674,-177.214,10.995,149.493
C06292=1115.372,353.970,-84.709,-177.210,10.998,149.493
C06293=1115.369,354.217,-84.745,-177.207,11.000,149.493
C06294=1115.365,354.465,-84.780,-177.203,11.002,149.493
C06295=1115.361,354.712,-84.816,-177.200,11.005,149.492
C06296=1115.358,354.960,-84.852,-177.197,11.007,149.492
C06297=1115.354,355.207,-84.887,-177.193,11.010,149.492
C06298=1115.350,355.453,-84.923,-177.190,11.013,149.492
C06299=1115.346,355.701,-84.959,-177.186,11.015,149.492
C06300=1115.342,355.949,-84.995,-177.182,11.017,149.491
C06301=1115.338,356.196,-85.030,-177.179,11.020,149.491
C06302=1115.335,356.444,-85.066,-177.176,11.022,149.491
C06303=1115.331,356.691,-85.101,-177.173,11.025,149.490
C06304=1115.327,356.939,-85.137,-177.169,11.027,149.490
C06305=1115.323,357.186,-85.173,-177.166,11.030,149.490
C06306=1115.320,357.433,-85.209,-177.162,11.032,149.490
C06307=1115.316,357.681,-85.245,-177.159,11.034,149.489
C06308=1115.312,357.928,-85.280,-177.156,11.037,149.489
C06309=1115.307,358.175,-85.316,-177.152,11.039,149.489
C06310=1115.304,358.422,-85.352,-177.149,11.042,149.489
C06311=1115.300,358.670,-85.388,-177.145,11.044,149.488
C06312=1115.297,358.917,-85.423,-177.142,11.046,149.488
C06313=1115.292,359.165,-85.460,-177.139,11.049,149.488
C06314=1115.289,359.412,-85.496,-177.135,11.051,149.488
C06315=1115.285,359.659,-85.531,-177.132,11.054,149.487
C06316=1115.281,359.907,-85.568,-177.128,11.056,149.487
C06317=1115.277,360.154,-85.604,-177.125,11.058,149.487
C06318=1115.274,360.402,-85.639,-177.122,11.061,149.487
C06319=1115.269,360.649,-85.676,-177.118,11.063,149.486
C06320=1115.266,360.896,-85.712,-177.115,11.065,149.486
C06321=1115.262,361.144,-85.747,-177.111,11.068,149.486
C06322=1115.258,361.391,-85.784,-177.108,11.070,149.486
C06323=1115.255,361.603,-85.814,-177.105,11.072,149.485
C06324=1115.252,361.815,-85.846,-177.103,11.074,149.485
C06325=1115.249,362.027,-85.877,-177.100,11.076,149.485
C06326=1115.245,362.239,-85.908,-177.097,11.078,149.485
C06327=1115.243,362.451,-85.938,-177.094,11.081,149.485
C06328=1115.239,362.663,-85.970,-177.091,11.082,149.484
C06329=1115.236,362.875,-86.001,-177.088,11.085,149.484
C06330=1115.232,363.087,-86.032,-177.085,11.087,149.484
C06331=1115.229,363.335,-86.068,-177.082,11.089,149.484
C06332=1115.226,363.582,-86.104,-177.078,11.091,149.483
C06333=1115.222,363.829,-86.141,-177.075,11.094,149.483
C06334=1115.218,364.076,-86.176,-177.072,11.096,149.483
C06335=1115.214,364.324,-86.213,-177.068,11.099,149.483
C06336=1115.210,364.571,-86.249,-177.065,11.101,149.482
C06337=1115.206,364.818,-86.286,-177.061,11.103,149.482
C06338=1115.203,365.065,-86.322,-177.058,11.106,149.482
C06339=1115.198,365.313,-86.358,-177.055,11.108,149.482
C06340=1115.195,365.560,-86.394,-177.051,11.111,149.481
C06341=1115.191,365.807,-86.431,-177.048,11.113,149.481
C06342=1115.187,366.055,-86.467,-177.045,11.115,149.481
C06343=1115.184,366.302,-86.504,-177.042,11.117,149.481
C06344=1115.180,366.549,-86.540,-177.038,11.119,149.480
C06345=1115.176,366.797,-86.577,-177.035,11.122,149.480
C06346=1115.172,367.044,-86.613,-177.032,11.124,149.480
C06347=1115.168,367.291,-86.649,-177.029,11.127,149.480
C06348=1115.164,367.538,-86.686,-177.025,11.129,149.479
C06349=1115.161,367.785,-86.723,-177.022,11.131,149.479
C06350=1115.157,368.032,-86.759,-177.018,11.134,149.479
C06351=1115.153,368.281,-86.796,-177.015,11.136,149.479
C06352=1115.150,368.528,-86.832,-177.012,11.139,149.478
C06353=1115.146,368.775,-86.869,-177.008,11.141,149.478
C06354=1115.142,369.022,-86.906,-177.005,11.144,149.478
C06355=1115.138,369.269,-86.942,-177.001,11.146,149.478
C06356=1115.134,369.516,-86.979,-176.998,11.148,149.477
C06357=1115.131,369.764,-87.016,-176.995,11.151,149.477
C06358=1115.127,370.011,-87.052,-176.991,11.153,149.477
C06359=1115.123,370.258,-87.089,-176.988,11.156,149.477
C06360=1115.119,370.505,-87.126,-176.985,11.158,149.477
C06361=1115.116,370.752,-87.162,-176.982,11.161,149.476
C06362=1115.112,371.000,-87.200,-176.978,11.163,149.476
C06363=1115.108,371.247,-87.237,-176.975,11.166,149.476
C06364=1115.105,371.494,-87.273,-176.972,11.168,149.476
C06365=1115.101,371.742,-87.310,-176.969,11.170,149.476
C06366=1115.097,371.989,-87.347,-176.966,11.172,149.475
C06367=1115.093,372.237,-87.384,-176.962,11.175,149.475
C06368=1115.090,372.483,-87.420,-176.959,11.177,149.475
C06369=1115.086,372.731,-87.457,-176.955,11.180,149.475
C06370=1115.082,372.979,-87.494,-176.952,11.182,149.474
C06371=1115.078,373.226,-87.531,-176.949,11.185,149.474
C06372=1115.074,373.473,-87.568,-176.946,11.187,149.474
C06373=1115.071,373.719,-87.605,-176.942,11.190,149.474
C06374=1115.067,373.967,-87.642,-176.939,11.192,149.474
C06375=1115.063,374.214,-87.679,-176.936,11.194,149.473
C06376=1115.059,374.461,-87.716,-176.932,11.197,149.473
C06377=1115.056,374.709,-87.753,-176.929,11.199,149.473
C06378=1115.052,374.956,-87.791,-176.926,11.202,149.473
C06379=1115.048,375.168,-87.821,-176.923,11.204,149.473
C06380=1115.046,375.380,-87.853,-176.920,11.206,149.472
C06381=1115.042,375.591,-87.885,-176.918,11.208,149.472
C06382=1115.039,375.803,-87.917,-176.915,11.211,149.472
C06383=1115.036,376.015,-87.949,-176.912,11.213,149.472
C06384=1115.033,376.227,-87.981,-176.910,11.215,149.472
C06385=1115.029,376.438,-88.013,-176.906,11.217,149.472
C06386=1115.027,376.650,-88.045,-176.904,11.219,149.471
C06387=1115.022,376.897,-88.082,-176.901,11.222,149.471
C06388=1115.018,377.145,-88.119,-176.898,11.224,149.471
C06389=1115.015,377.392,-88.157,-176.894,11.227,149.471
C06390=1115.011,377.639,-88.193,-176.891,11.229,149.471
C06391=1115.008,377.887,-88.231,-176.888,11.232,149.471
C06392=1115.004,378.134,-88.268,-176.884,11.234,149.470
C06393=1115.000,378.381,-88.305,-176.881,11.237,149.470
C06394=1114.997,378.628,-88.343,-176.878,11.239,149.470
C06395=1114.992,378.875,-88.380,-176.875,11.242,149.470
C06396=1114.989,379.122,-88.417,-176.872,11.244,149.470
C06397=1114.985,379.370,-88.455,-176.869,11.247,149.470
C06398=1114.981,379.616,-88.492,-176.865,11.250,149.470
C06399=1114.978,379.864,-88.529,-176.862,11.252,149.469
C06400=1114.974,380.111,-88.567,-176.859,11.255,149.469
C06401=1114.970,380.358,-88.604,-176.856,11.257,149.469
C06402=1114.967,380.605,-88.642,-176.853,11.260,149.469
C06403=1114.963,380.852,-88.679,-176.850,11.263,149.469
C06404=1114.960,381.100,-88.717,-176.846,11.265,149.469
C06405=1114.956,381.346,-88.754,-176.843,11.268,149.469
C06406=1114.952,381.594,-88.791,-176.840,11.271,149.469
C06407=1114.948,381.841,-88.829,-176.837,11.273,149.468
C06408=1114.945,382.088,-88.867,-176.834,11.275,149.468
C06409=1114.941,382.335,-88.904,-176.831,11.278,149.468
C06410=1114.937,382.582,-88.942,-176.827,11.281,149.468
C06411=1114.933,382.829,-88.980,-176.825,11.284,149.468
C06412=1114.929,383.076,-89.017,-176.821,11.286,149.468
C06413=1114.926,383.324,-89.055,-176.818,11.289,149.468
C06414=1114.922,383.570,-89.092,-176.815,11.292,149.468
C06415=1114.919,383.818,-89.130,-176.813,11.294,149.468
C06416=1114.915,384.065,-89.167,-176.810,11.297,149.468
C06417=1114.911,384.312,-89.206,-176.808,11.299,149.468
C06418=1114.907,384.559,-89.243,-176.805,11.301,149.468
C06419=1114.904,384.806,-89.281,-176.803,11.303,149.468
C06420=1114.900,385.053,-89.319,-176.801,11.305,149.468
C06421=1114.897,385.301,-89.356,-176.798,11.309,149.468
C06422=1114.892,385.548,-89.394,-176.796,11.311,149.468
C06423=1114.889,385.795,-89.432,-176.793,11.313,149.468
C06424=1114.886,386.042,-89.470,-176.791,11.316,149.468
C06425=1114.882,386.289,-89.508,-176.788,11.319,149.468
C06426=1114.878,386.536,-89.546,-176.786,11.321,149.468
C06427=1114.875,386.783,-89.584,-176.783,11.324,149.468
C06428=1114.871,387.030,-89.622,-176.781,11.326,149.468
C06429=1114.867,387.277,-89.658,-176.779,11.329,149.468
C06430=1114.863,387.525,-89.697,-176.776,11.331,149.468
C06431=1114.860,387.771,-89.735,-176.774,11.334,149.468
C06432=1114.856,388.019,-89.772,-176.771,11.337,149.468
C06433=1114.853,388.266,-89.810,-176.769,11.339,149.468
C06434=1114.849,388.513,-89.849,-176.767,11.343,149.469
C06435=1114.846,388.724,-89.881,-176.765,11.345,149.469
C06436=1114.843,388.937,-89.914,-176.763,11.347,149.469
C06437=1114.840,389.147,-89.946,-176.761,11.350,149.469
C06438=1114.836,389.360,-89.979,-176.759,11.352,149.469
C06439=1114.834,389.571,-90.012,-176.757,11.354,149.469
C06440=1114.830,389.783,-90.044,-176.755,11.356,149.469
C06441=1114.827,389.994,-90.076,-176.752,11.359,149.469
C06442=1114.824,390.206,-90.110,-176.751,11.362,149.469
C06443=1114.821,390.453,-90.148,-176.749,11.364,149.470
C06444=1114.817,390.700,-90.185,-176.747,11.368,149.470
C06445=1114.813,390.947,-90.224,-176.744,11.371,149.470
C06446=1114.809,391.194,-90.261,-176.742,11.374,149.470
C06447=1114.806,391.441,-90.299,-176.740,11.376,149.470
C06448=1114.802,391.689,-90.338,-176.737,11.379,149.471
C06449=1114.799,391.935,-90.375,-176.735,11.383,149.471
C06450=1114.795,392.182,-90.415,-176.733,11.386,149.471
C06451=1114.792,392.429,-90.453,-176.730,11.389,149.471
C06452=1114.788,392.676,-90.490,-176.729,11.392,149.472
C06453=1114.784,392.924,-90.529,-176.726,11.395,149.472
C06454=1114.781,393.171,-90.567,-176.724,11.399,149.472
C06455=1114.777,393.417,-90.606,-176.722,11.402,149.472
C06456=1114.773,393.664,-90.643,-176.719,11.405,149.473
C06457=1114.769,393.912,-90.682,-176.717,11.409,149.473
C06458=1114.766,394.158,-90.720,-176.715,11.412,149.473
C06459=1114.762,394.405,-90.759,-176.713,11.415,149.474
C06460=1114.759,394.653,-90.797,-176.711,11.419,149.474
C06461=1114.754,394.900,-90.835,-176.708,11.422,149.474
C06462=1114.751,395.146,-90.874,-176.707,11.425,149.475
C06463=1114.748,395.394,-90.912,-176.705,11.428,149.475
C06464=1114.744,395.641,-90.950,-176.702,11.432,149.475
C06465=1114.740,395.887,-90.989,-176.700,11.435,149.476
C06466=1114.737,396.135,-91.027,-176.698,11.439,149.476
C06467=1114.733,396.382,-91.066,-176.696,11.443,149.477
C06468=1114.730,396.628,-91.104,-176.694,11.447,149.477
C06469=1114.726,396.876,-91.142,-176.692,11.450,149.477
C06470=1114.723,397.122,-91.181,-176.690,11.453,149.478
C06471=1114.719,397.370,-91.219,-176.688,11.457,149.478
C06472=1114.715,397.616,-91.258,-176.686,11.461,149.479
C06473=1114.711,397.864,-91.296,-176.684,11.464,149.479
C06474=1114.708,398.110,-91.336,-176.682,11.468,149.480
C06475=1114.705,398.358,-91.373,-176.679,11.472,149.480
C06476=1114.700,398.604,-91.412,-176.677,11.476,149.481
C06477=1114.697,398.851,-91.450,-176.675,11.480,149.481
C06478=1114.694,399.098,-91.490,-176.674,11.483,149.482
C06479=1114.690,399.346,-91.528,-176.672,11.487,149.482
C06480=1114.687,399.592,-91.567,-176.670,11.492,149.483
C06481=1114.682,399.839,-91.605,-176.667,11.495,149.483
C06482=1114.679,400.086,-91.644,-176.666,11.499,149.484
C06483=1114.676,400.333,-91.683,-176.663,11.504,149.484
C06484=1114.672,400.581,-91.721,-176.662,11.507,149.485
C06485=1114.668,400.828,-91.761,-176.660,11.511,149.485
C06486=1114.665,401.073,-91.799,-176.658,11.516,149.486
C06487=1114.661,401.321,-91.837,-176.656,11.520,149.487
C06488=1114.657,401.568,-91.877,-176.655,11.524,149.487
C06489=1114.654,401.815,-91.915,-176.652,11.528,149.488
C06490=1114.650,402.062,-91.954,-176.650,11.532,149.488
C06491=1114.647,402.274,-91.987,-176.649,11.536,149.489
C06492=1114.644,402.485,-92.021,-176.647,11.540,149.490
C06493=1114.641,402.696,-92.054,-176.645,11.543,149.490
C06494=1114.638,402.907,-92.087,-176.644,11.546,149.491
C06495=1114.635,403.119,-92.120,-176.643,11.551,149.491
C06496=1114.632,403.331,-92.153,-176.641,11.554,149.492
C06497=1114.629,403.543,-92.187,-176.639,11.558,149.492
C06498=1114.626,403.754,-92.221,-176.638,11.562,149.493
C06499=1114.622,404.001,-92.259,-176.636,11.566,149.494
C06500=1114.619,404.248,-92.298,-176.634,11.571,149.495
C06501=1114.615,404.495,-92.337,-176.632,11.576,149.495
C06502=1114.612,404.742,-92.376,-176.631,11.580,149.496
C06503=1114.608,404.988,-92.415,-176.629,11.585,149.497
C06504=1114.605,405.235,-92.454,-176.627,11.590,149.498
C06505=1114.601,405.482,-92.493,-176.626,11.594,149.498
C06506=1114.597,405.729,-92.532,-176.624,11.599,149.499
C06507=1114.593,405.976,-92.571,-176.622,11.604,149.500
C06508=1114.590,406.223,-92.610,-176.621,11.608,149.501
C06509=1114.586,406.470,-92.649,-176.619,11.613,149.502
C06510=1114.583,406.717,-92.688,-176.617,11.618,149.502
C06511=1114.580,406.964,-92.727,-176.615,11.623,149.503
C06512=1114.576,407.211,-92.767,-176.614,11.627,149.504
C06513=1114.572,407.458,-92.806,-176.612,11.632,149.505
C06514=1114.569,407.705,-92.845,-176.611,11.637,149.506
C06515=1114.565,407.952,-92.884,-176.609,11.643,149.507
C06516=1114.562,408.199,-92.924,-176.607,11.648,149.508
C06517=1114.558,408.446,-92.963,-176.606,11.653,149.509
C06518=1114.555,408.692,-93.002,-176.604,11.658,149.510
C06519=1114.552,408.939,-93.042,-176.603,11.662,149.511
C06520=1114.548,409.185,-93.081,-176.601,11.668,149.512
C06521=1114.545,409.432,-93.120,-176.600,11.673,149.513
C06522=1114.541,409.679,-93.159,-176.598,11.678,149.514
C06523=1114.537,409.926,-93.199,-176.597,11.684,149.515
C06524=1114.534,410.173,-93.238,-176.595,11.689,149.516
C06525=1114.530,410.420,-93.277,-176.594,11.694,149.517
C06526=1114.527,410.667,-93.317,-176.592,11.700,149.518
C06527=1114.523,410.914,-93.356,-176.590,11.706,149.519
C06528=1114.520,411.161,-93.395,-176.589,11.711,149.520
C06529=1114.516,411.408,-93.435,-176.588,11.716,149.521
C06530=1114.512,411.654,-93.474,-176.586,11.722,149.522
C06531=1114.509,411.901,-93.514,-176.585,11.727,149.523
C06532=1114.505,412.148,-93.553,-176.584,11.733,149.524
C06533=1114.502,412.395,-93.592,-176.582,11.739,149.525
C06534=1114.498,412.641,-93.632,-176.581,11.745,149.527
C06535=1114.495,412.888,-93.672,-176.579,11.750,149.528
C06536=1114.491,413.135,-93.711,-176.578,11.756,149.529
C06537=1114.488,413.381,-93.751,-176.576,11.762,149.530
C06538=1114.485,413.629,-93.790,-176.575,11.768,149.531
C06539=1114.482,413.875,-93.830,-176.574,11.773,149.533
C06540=1114.479,414.123,-93.869,-176.573,11.779,149.534
C06541=1114.477,414.369,-93.909,-176.571,11.785,149.535
C06542=1114.476,414.616,-93.948,-176.571,11.791,149.536
C06543=1114.475,414.863,-93.988,-176.569,11.798,149.537
C06544=1114.476,415.110,-94.027,-176.568,11.803,149.539
C06545=1114.476,415.357,-94.066,-176.567,11.809,149.540
C06546=1114.476,415.604,-94.105,-176.566,11.816,149.541
C06547=1114.477,415.815,-94.139,-176.565,11.821,149.543
C06548=1114.479,416.026,-94.172,-176.564,11.826,149.544
C06549=1114.481,416.238,-94.204,-176.563,11.832,149.545
C06550=1114.483,416.449,-94.238,-176.562,11.837,149.546
C06551=1114.485,416.660,-94.271,-176.561,11.842,149.547
C06552=1114.488,416.871,-94.305,-176.561,11.847,149.548
C06553=1114.492,417.082,-94.338,-176.559,11.853,149.550
C06554=1114.496,417.294,-94.371,-176.559,11.859,149.551
C06555=1114.077,417.293,-94.433,-176.551,11.863,149.550
C06556=1114.073,417.082,-94.401,-176.552,11.857,149.549
C06557=1114.069,416.871,-94.368,-176.553,11.852,149.548
C06558=1114.066,416.660,-94.335,-176.553,11.846,149.546
C06559=1114.064,416.449,-94.301,-176.555,11.841,149.545
C06560=1114.062,416.238,-94.267,-176.556,11.835,149.544
C06561=1114.060,416.026,-94.234,-176.556,11.831,149.543
C06562=1114.058,415.815,-94.201,-176.558,11.825,149.542
C06563=1114.057,415.603,-94.167,-176.559,11.819,149.541
C06564=1114.057,415.357,-94.128,-176.560,11.814,149.539
C06565=1114.057,415.110,-94.090,-176.561,11.808,149.538
C06566=1114.056,414.864,-94.050,-176.562,11.801,149.537
C06567=1114.057,414.616,-94.010,-176.563,11.796,149.536
C06568=1114.058,414.369,-93.972,-176.565,11.789,149.534
C06569=1114.060,414.122,-93.932,-176.566,11.783,149.533
C06570=1114.062,413.876,-93.892,-176.568,11.777,149.532
C06571=1114.065,413.628,-93.853,-176.569,11.771,149.531
C06572=1114.069,413.382,-93.813,-176.570,11.766,149.529
C06573=1114.072,413.135,-93.774,-176.572,11.760,149.528
C06574=1114.076,412.888,-93.734,-176.573,11.754,149.527
C06575=1114.079,412.642,-93.694,-176.574,11.749,149.526
C06576=1114.083,412.395,-93.655,-176.576,11.742,149.525
C06577=1114.086,412.147,-93.616,-176.577,11.737,149.524
C06578=1114.089,411.901,-93.576,-176.579,11.731,149.522
C06579=1114.093,411.654,-93.536,-176.580,11.726,149.521
C06580=1114.096,411.407,-93.497,-176.582,11.720,149.520
C06581=1114.100,411.160,-93.457,-176.584,11.714,149.519
C06582=1114.103,410.914,-93.418,-176.585,11.709,149.518
C06583=1114.107,410.667,-93.379,-176.586,11.704,149.517
C06584=1114.111,410.420,-93.339,-176.588,11.698,149.516
C06585=1114.114,410.173,-93.299,-176.589,11.693,149.515
C06586=1114.117,409.926,-93.260,-176.591,11.688,149.514
C06587=1114.121,409.679,-93.221,-176.592,11.682,149.513
C06588=1114.125,409.432,-93.182,-176.594,11.677,149.512
C06589=1114.128,409.185,-93.142,-176.595,11.672,149.511
C06590=1114.132,408.938,-93.103,-176.597,11.667,149.510
C06591=1114.136,408.691,-93.064,-176.599,11.661,149.509
C06592=1114.139,408.445,-93.025,-176.600,11.656,149.508
C06593=1114.143,408.198,-92.985,-176.602,11.651,149.507
C06594=1114.146,407.951,-92.945,-176.604,11.646,149.506
C06595=1114.150,407.704,-92.906,-176.605,11.641,149.506
C06596=1114.153,407.458,-92.868,-176.607,11.636,149.505
C06597=1114.156,407.211,-92.828,-176.609,11.631,149.504
C06598=1114.160,406.964,-92.789,-176.610,11.625,149.503
C06599=1114.163,406.717,-92.750,-176.612,11.621,149.502
C06600=1114.167,406.470,-92.711,-176.614,11.616,149.501
C06601=1114.171,406.223,-92.671,-176.615,11.611,149.500
C06602=1114.174,405.976,-92.632,-176.617,11.606,149.499
C06603=1114.177,405.729,-92.593,-176.619,11.601,149.499
C06604=1114.181,405.482,-92.554,-176.621,11.597,149.498
C06605=1114.185,405.235,-92.516,-176.623,11.592,149.497
C06606=1114.189,404.988,-92.477,-176.624,11.587,149.496
C06607=1114.193,404.741,-92.437,-176.626,11.583,149.496
C06608=1114.195,404.495,-92.399,-176.628,11.578,149.495
C06609=1114.199,404.248,-92.360,-176.630,11.574,149.494
C06610=1114.203,404.001,-92.320,-176.632,11.569,149.493
C06611=1114.206,403.754,-92.281,-176.633,11.565,149.493
C06612=1114.210,403.542,-92.248,-176.635,11.561,149.492
C06613=1114.212,403.331,-92.215,-176.636,11.557,149.491
C06614=1114.215,403.119,-92.182,-176.638,11.553,149.491
C06615=1114.219,402.909,-92.148,-176.640,11.549,149.490
C06616=1114.222,402.697,-92.115,-176.642,11.546,149.490
C06617=1114.225,402.485,-92.082,-176.643,11.542,149.489
C06618=1114.228,402.274,-92.048,-176.645,11.538,149.489
C06619=1114.231,402.062,-92.015,-176.646,11.535,149.488
C06620=1114.234,401.815,-91.976,-176.649,11.530,149.488
C06621=1114.238,401.568,-91.937,-176.650,11.526,149.487
C06622=1114.242,401.321,-91.898,-176.652,11.522,149.486
C06623=1114.245,401.075,-91.860,-176.654,11.518,149.486
C06624=1114.249,400.828,-91.821,-176.656,11.513,149.485
C06625=1114.253,400.580,-91.782,-176.658,11.510,149.484
C06626=1114.256,400.333,-91.744,-176.660,11.506,149.484
C06627=1114.259,400.087,-91.704,-176.662,11.501,149.483
C06628=1114.264,399.840,-91.666,-176.664,11.497,149.483
C06629=1114.267,399.593,-91.628,-176.666,11.494,149.482
C06630=1114.271,399.345,-91.589,-176.668,11.489,149.482
C06631=1114.274,399.098,-91.550,-176.670,11.485,149.481
C06632=1114.277,398.851,-91.512,-176.672,11.482,149.481
C06633=1114.282,398.605,-91.473,-176.674,11.477,149.480
C06634=1114.284,398.358,-91.434,-176.676,11.474,149.480
C06635=1114.288,398.111,-91.396,-176.678,11.470,149.479
C06636=1114.292,397.864,-91.357,-176.680,11.467,149.479
C06637=1114.296,397.617,-91.319,-176.682,11.463,149.478
C06638=1114.299,397.370,-91.280,-176.685,11.459,149.478
C06639=1114.303,397.123,-91.242,-176.687,11.455,149.478
C06640=1114.307,396.875,-91.203,-176.689,11.452,149.477
C06641=1114.310,396.629,-91.165,-176.691,11.448,149.477
C06642=1114.314,396.382,-91.126,-176.693,11.444,149.476
C06643=1114.318,396.135,-91.087,-176.695,11.441,149.476
C06644=1114.321,395.888,-91.049,-176.697,11.437,149.476
C06645=1114.325,395.641,-91.011,-176.699,11.434,149.475
C06646=1114.328,395.394,-90.972,-176.701,11.431,149.475
C06647=1114.332,395.146,-90.934,-176.703,11.427,149.474
C06648=1114.335,394.900,-90.895,-176.705,11.424,149.474
C06649=1114.339,394.653,-90.857,-176.708,11.420,149.474
C06650=1114.343,394.406,-90.819,-176.710,11.417,149.474
C06651=1114.347,394.158,-90.781,-176.712,11.413,149.473
C06652=1114.350,393.912,-90.742,-176.715,11.410,149.473
C06653=1114.354,393.665,-90.704,-176.717,11.407,149.473
C06654=1114.357,393.417,-90.666,-176.719,11.403,149.472
C06655=1114.361,393.171,-90.628,-176.721,11.400,149.472
C06656=1114.365,392.924,-90.589,-176.723,11.397,149.472
C06657=1114.368,392.676,-90.551,-176.726,11.394,149.471
C06658=1114.372,392.430,-90.513,-176.728,11.390,149.471
C06659=1114.375,392.182,-90.475,-176.731,11.387,149.471
C06660=1114.379,391.935,-90.436,-176.733,11.384,149.471
C06661=1114.383,391.689,-90.398,-176.735,11.382,149.471
C06662=1114.386,391.442,-90.360,-176.737,11.378,149.470
C06663=1114.390,391.194,-90.322,-176.740,11.375,149.470
C06664=1114.394,390.947,-90.284,-176.742,11.372,149.470
C06665=1114.397,390.700,-90.246,-176.745,11.369,149.470
C06666=1114.402,390.453,-90.208,-176.746,11.366,149.470
C06667=1114.404,390.207,-90.169,-176.749,11.363,149.469
C06668=1114.408,389.994,-90.137,-176.751,11.361,149.469
C06669=1114.410,389.783,-90.104,-176.753,11.358,149.469
C06670=1114.414,389.571,-90.072,-176.755,11.355,149.469
C06671=1114.417,389.360,-90.039,-176.757,11.353,149.469
C06672=1114.420,389.147,-90.007,-176.759,11.351,149.469
C06673=1114.423,388.937,-89.974,-176.761,11.348,149.469
C06674=1114.427,388.724,-89.942,-176.763,11.346,149.469
C06675=1114.429,388.513,-89.909,-176.765,11.344,149.468
C06676=1114.433,388.266,-89.871,-176.767,11.341,149.468
C06677=1114.437,388.019,-89.833,-176.770,11.337,149.468
C06678=1114.441,387.772,-89.795,-176.772,11.335,149.468
C06679=1114.444,387.525,-89.757,-176.775,11.332,149.468
C06680=1114.448,387.277,-89.719,-176.777,11.330,149.468
C06681=1114.452,387.031,-89.681,-176.779,11.327,149.468
C06682=1114.455,386.784,-89.643,-176.782,11.324,149.468
C06683=1114.459,386.537,-89.606,-176.784,11.322,149.468
C06684=1114.463,386.289,-89.568,-176.787,11.319,149.468
C06685=1114.467,386.042,-89.530,-176.789,11.317,149.468
C06686=1114.470,385.795,-89.492,-176.792,11.314,149.468
C06687=1114.474,385.548,-89.455,-176.794,11.312,149.468
C06688=1114.477,385.301,-89.417,-176.797,11.309,149.468
C06689=1114.481,385.054,-89.378,-176.799,11.307,149.467
C06690=1114.484,384.807,-89.341,-176.802,11.304,149.467
C06691=1114.488,384.559,-89.303,-176.804,11.302,149.468
C06692=1114.492,384.313,-89.266,-176.806,11.300,149.468
C06693=1114.495,384.065,-89.228,-176.809,11.297,149.468
C06694=1114.499,383.818,-89.190,-176.812,11.295,149.468
C06695=1114.503,383.571,-89.152,-176.814,11.292,149.468
C06696=1114.507,383.324,-89.115,-176.817,11.290,149.468
C06697=1114.510,383.077,-89.077,-176.820,11.287,149.468
C06698=1114.514,382.830,-89.040,-176.824,11.284,149.468
C06699=1114.518,382.583,-89.003,-176.827,11.282,149.468
C06700=1114.521,382.336,-88.965,-176.830,11.279,149.468
C06701=1114.526,382.089,-88.927,-176.833,11.276,149.468
C06702=1114.529,381.842,-88.889,-176.836,11.273,149.468
C06703=1114.533,381.594,-88.852,-176.839,11.271,149.468
C06704=1114.536,381.347,-88.814,-176.842,11.268,149.468
C06705=1114.540,381.100,-88.777,-176.845,11.266,149.469
C06706=1114.543,380.853,-88.739,-176.849,11.263,149.469
C06707=1114.547,380.606,-88.701,-176.852,11.260,149.469
C06708=1114.551,380.358,-88.664,-176.855,11.258,149.469
C06709=1114.554,380.112,-88.627,-176.858,11.255,149.469
C06710=1114.558,379.864,-88.590,-176.861,11.253,149.469
C06711=1114.562,379.617,-88.552,-176.864,11.250,149.469
C06712=1114.566,379.370,-88.515,-176.868,11.248,149.470
C06713=1114.569,379.123,-88.477,-176.871,11.245,149.470
C06714=1114.573,378.875,-88.440,-176.874,11.242,149.470
C06715=1114.577,378.629,-88.403,-176.877,11.240,149.470
C06716=1114.580,378.381,-88.365,-176.880,11.237,149.470
C06717=1114.584,378.134,-88.328,-176.884,11.235,149.470
C06718=1114.588,377.887,-88.291,-176.887,11.232,149.471
C06719=1114.591,377.640,-88.253,-176.890,11.230,149.471
C06720=1114.595,377.393,-88.216,-176.893,11.227,149.471
C06721=1114.599,377.145,-88.179,-176.897,11.225,149.471
C06722=1114.603,376.898,-88.141,-176.900,11.222,149.471
C06723=1114.607,376.651,-88.104,-176.903,11.220,149.471
C06724=1114.610,376.439,-88.073,-176.906,11.218,149.472
C06725=1114.613,376.228,-88.041,-176.909,11.215,149.472
C06726=1114.616,376.015,-88.008,-176.911,11.213,149.472
C06727=1114.620,375.804,-87.977,-176.914,11.211,149.472
C06728=1114.623,375.591,-87.945,-176.917,11.209,149.472
C06729=1114.626,375.380,-87.914,-176.920,11.207,149.472
C06730=1114.629,375.168,-87.882,-176.922,11.204,149.473
C06731=1114.632,374.957,-87.850,-176.925,11.203,149.473
C06732=1114.636,374.710,-87.813,-176.928,11.200,149.473
C06733=1114.639,374.462,-87.775,-176.932,11.198,149.473
C06734=1114.644,374.215,-87.738,-176.935,11.195,149.473
C06735=1114.648,373.968,-87.702,-176.938,11.193,149.474
C06736=1114.651,373.721,-87.665,-176.942,11.190,149.474
C06737=1114.655,373.473,-87.628,-176.945,11.188,149.474
C06738=1114.659,373.226,-87.591,-176.948,11.185,149.474
C06739=1114.662,372.979,-87.554,-176.952,11.183,149.474
C06740=1114.666,372.732,-87.516,-176.955,11.180,149.475
C06741=1114.669,372.485,-87.480,-176.958,11.178,149.475
C06742=1114.673,372.237,-87.443,-176.961,11.175,149.475
C06743=1114.677,371.990,-87.407,-176.965,11.173,149.475
C06744=1114.681,371.742,-87.369,-176.968,11.170,149.475
C06745=1114.684,371.495,-87.333,-176.971,11.168,149.476
C06746=1114.688,371.248,-87.296,-176.975,11.165,149.476
C06747=1114.692,371.001,-87.259,-176.978,11.163,149.476
C06748=1114.697,370.754,-87.222,-176.981,11.161,149.476
C06749=1114.699,370.506,-87.186,-176.984,11.158,149.476
C06750=1114.703,370.259,-87.149,-176.988,11.156,149.477
C06751=1114.708,370.012,-87.112,-176.991,11.153,149.477
C06752=1114.711,369.765,-87.076,-176.995,11.151,149.477
C06753=1114.715,369.518,-87.039,-176.998,11.148,149.477
C06754=1114.718,369.270,-87.002,-177.001,11.147,149.478
C06755=1114.722,369.023,-86.965,-177.004,11.144,149.478
C06756=1114.726,368.776,-86.929,-177.007,11.142,149.478
C06757=1114.730,368.528,-86.892,-177.011,11.139,149.478
C06758=1114.734,368.281,-86.856,-177.014,11.137,149.479
C06759=1114.738,368.034,-86.819,-177.018,11.135,149.479
C06760=1114.741,367.786,-86.783,-177.021,11.132,149.479
C06761=1114.745,367.539,-86.746,-177.024,11.130,149.479
C06762=1114.749,367.292,-86.709,-177.028,11.127,149.480
C06763=1114.752,367.045,-86.673,-177.031,11.125,149.480
C06764=1114.756,366.797,-86.637,-177.035,11.123,149.480
C06765=1114.760,366.551,-86.600,-177.038,11.120,149.480
C06766=1114.764,366.303,-86.563,-177.041,11.118,149.481
C06767=1114.768,366.056,-86.527,-177.044,11.115,149.481
C06768=1114.771,365.808,-86.491,-177.048,11.113,149.481
C06769=1114.775,365.561,-86.454,-177.051,11.110,149.481
C06770=1114.779,365.313,-86.418,-177.055,11.108,149.482
C06771=1114.783,365.066,-86.381,-177.058,11.106,149.482
C06772=1114.786,364.819,-86.345,-177.061,11.103,149.482
C06773=1114.791,364.571,-86.309,-177.065,11.101,149.482
C06774=1114.794,364.324,-86.273,-177.068,11.098,149.482
C06775=1114.798,364.077,-86.236,-177.072,11.096,149.483
C06776=1114.802,363.830,-86.200,-177.075,11.094,149.483
C06777=1114.806,363.583,-86.164,-177.078,11.091,149.483
C06778=1114.810,363.335,-86.128,-177.082,11.089,149.483
C06779=1114.813,363.088,-86.092,-177.085,11.087,149.484
C06780=1114.816,362.876,-86.060,-177.088,11.085,149.484
C06781=1114.820,362.664,-86.030,-177.090,11.083,149.484
C06782=1114.823,362.452,-85.999,-177.094,11.080,149.484
C06783=1114.825,362.240,-85.967,-177.096,11.079,149.485
C06784=1114.829,362.028,-85.936,-177.100,11.076,149.485
C06785=1114.833,361.816,-85.905,-177.102,11.075,149.485
C06786=1114.835,361.604,-85.875,-177.105,11.073,149.485
C06787=1114.838,361.392,-85.844,-177.108,11.070,149.486
C06788=1114.843,361.145,-85.807,-177.111,11.068,149.486
C06789=1114.846,360.897,-85.771,-177.115,11.065,149.486
C06790=1114.850,360.650,-85.736,-177.118,11.063,149.486
C06791=1114.854,360.402,-85.699,-177.122,11.061,149.487
C06792=1114.858,360.155,-85.663,-177.125,11.058,149.487
C06793=1114.861,359.908,-85.627,-177.128,11.056,149.487
C06794=1114.865,359.660,-85.591,-177.132,11.053,149.487
C06795=1114.869,359.413,-85.556,-177.135,11.051,149.488
C06796=1114.872,359.166,-85.519,-177.139,11.049,149.488
C06797=1114.877,358.919,-85.484,-177.142,11.046,149.488
C06798=1114.881,358.671,-85.448,-177.145,11.044,149.488
C06799=1114.885,358.424,-85.412,-177.149,11.041,149.489
C06800=1114.888,358.177,-85.376,-177.152,11.039,149.489
C06801=1114.892,357.929,-85.341,-177.156,11.037,149.489
C06802=1114.896,357.682,-85.304,-177.159,11.034,149.489
C06803=1114.900,357.434,-85.269,-177.162,11.032,149.490
C06804=1114.904,357.187,-85.233,-177.166,11.029,149.490
C06805=1114.907,356.940,-85.197,-177.169,11.027,149.490
C06806=1114.911,356.692,-85.161,-177.173,11.025,149.490
C06807=1114.915,356.444,-85.125,-177.176,11.022,149.491
C06808=1114.919,356.197,-85.090,-177.179,11.020,149.491
C06809=1114.922,355.949,-85.054,-177.182,11.017,149.491
C06810=1114.927,355.703,-85.019,-177.186,11.015,149.491
C06811=1114.930,355.455,-84.984,-177.189,11.012,149.492
C06812=1114.935,355.207,-84.947,-177.193,11.010,149.492
C06813=1114.938,354.960,-84.912,-177.196,11.008,149.492
C06814=1114.942,354.713,-84.876,-177.199,11.005,149.492
C06815=1114.945,354.465,-84.840,-177.203,11.003,149.493
C06816=1114.949,354.218,-84.804,-177.206,11.000,149.493
C06817=1114.953,353.971,-84.769,-177.209,10.998,149.493
C06818=1114.957,353.724,-84.734,-177.213,10.996,149.493
C06819=1114.961,353.476,-84.698,-177.216,10.993,149.494
C06820=1114.964,353.228,-84.663,-177.220,10.991,149.494
C06821=1114.969,352.980,-84.627,-177.223,10.988,149.494
C06822=1114.973,352.733,-84.592,-177.226,10.986,149.494
C06823=1114.977,352.486,-84.557,-177.230,10.984,149.495
C06824=1114.980,352.238,-84.521,-177.234,10.980,149.495
C06825=1114.984,351.991,-84.485,-177.237,10.978,149.495
C06826=1114.988,351.743,-84.450,-177.240,10.975,149.495
C06827=1114.991,351.496,-84.414,-177.243,10.973,149.495
C06828=1114.996,351.248,-84.380,-177.247,10.970,149.496
C06829=1115.000,351.001,-84.344,-177.250,10.968,149.496
C06830=1115.003,350.753,-84.309,-177.253,10.966,149.496
C06831=1115.007,350.506,-84.273,-177.257,10.963,149.496
C06832=1115.011,350.259,-84.238,-177.260,10.961,149.497
C06833=1115.015,350.011,-84.203,-177.264,10.958,149.497
C06834=1115.019,349.764,-84.168,-177.267,10.956,149.497
C06835=1115.023,349.516,-84.132,-177.271,10.953,149.497
C06836=1115.026,349.304,-84.102,-177.273,10.951,149.498
C06837=1115.029,349.092,-84.072,-177.276,10.949,149.498
C06838=1115.033,348.880,-84.042,-177.279,10.946,149.498
C06839=1115.036,348.668,-84.012,-177.282,10.945,149.498
C06840=1115.039,348.456,-83.982,-177.284,10.943,149.498
C06841=1115.042,348.244,-83.951,-177.287,10.940,149.498
C06842=1115.046,348.031,-83.922,-177.290,10.938,149.499
C06843=1115.049,347.819,-83.892,-177.292,10.936,149.499
C06844=1115.053,347.572,-83.857,-177.295,10.934,149.499
C06845=1115.057,347.325,-83.821,-177.299,10.932,149.499
C06846=1115.061,347.077,-83.786,-177.302,10.929,149.499
C06847=1115.064,346.829,-83.751,-177.305,10.927,149.500
C06848=1115.069,346.582,-83.716,-177.308,10.924,149.500
C06849=1115.073,346.334,-83.681,-177.312,10.921,149.500
C06850=1115.077,346.087,-83.646,-177.315,10.919,149.500
C06851=1115.080,345.840,-83.611,-177.318,10.916,149.500
C06852=1115.084,345.592,-83.577,-177.322,10.914,149.501
C06853=1115.088,345.345,-83.541,-177.325,10.912,149.501
C06854=1115.092,345.097,-83.507,-177.327,10.910,149.501
C06855=1115.096,344.849,-83.471,-177.330,10.907,149.501
C06856=1115.100,344.602,-83.437,-177.334,10.905,149.501
C06857=1115.103,344.355,-83.402,-177.337,10.902,149.502
C06858=1115.107,344.107,-83.367,-177.340,10.900,149.502
C06859=1115.112,343.859,-83.332,-177.343,10.897,149.502
C06860=1115.115,343.612,-83.297,-177.347,10.894,149.502
C06861=1115.120,343.364,-83.263,-177.350,10.892,149.502
C06862=1115.123,343.116,-83.228,-177.353,10.890,149.503
C06863=1115.127,342.869,-83.193,-177.357,10.887,149.503
C06864=1115.131,342.622,-83.159,-177.359,10.884,149.503
C06865=1115.135,342.374,-83.124,-177.363,10.882,149.503
C06866=1115.139,342.127,-83.089,-177.365,10.880,149.503
C06867=1115.143,341.879,-83.054,-177.369,10.878,149.504
C06868=1115.147,341.632,-83.020,-177.372,10.875,149.504
C06869=1115.151,341.383,-82.985,-177.375,10.872,149.504
C06870=1115.155,341.137,-82.950,-177.378,10.870,149.504
C06871=1115.158,340.889,-82.916,-177.382,10.868,149.504
C06872=1115.162,340.641,-82.881,-177.385,10.865,149.505
C06873=1115.167,340.393,-82.846,-177.388,10.863,149.505
C06874=1115.170,340.146,-82.812,-177.391,10.860,149.505
C06875=1115.175,339.899,-82.777,-177.394,10.857,149.505
C06876=1115.178,339.651,-82.743,-177.398,10.855,149.505
C06877=1115.182,339.403,-82.708,-177.401,10.853,149.506
C06878=1115.186,339.155,-82.673,-177.403,10.850,149.506
C06879=1115.190,338.908,-82.640,-177.407,10.848,149.506
C06880=1115.194,338.660,-82.605,-177.410,10.846,149.506
C06881=1115.198,338.413,-82.571,-177.413,10.843,149.506
C06882=1115.202,338.165,-82.536,-177.416,10.840,149.506
C06883=1115.206,337.917,-82.502,-177.420,10.838,149.507
C06884=1115.210,337.670,-82.468,-177.423,10.835,149.507
C06885=1115.214,337.422,-82.433,-177.426,10.833,149.507
C06886=1115.218,337.175,-82.399,-177.429,10.830,149.507
C06887=1115.222,336.927,-82.364,-177.432,10.828,149.507
C06888=1115.226,336.680,-82.330,-177.436,10.825,149.508
C06889=1115.230,336.432,-82.295,-177.438,10.824,149.508
C06890=1115.234,336.185,-82.262,-177.441,10.821,149.508
C06891=1115.238,335.937,-82.227,-177.445,10.818,149.508
C06892=1115.241,335.724,-82.197,-177.448,10.816,149.508
C06893=1115.245,335.513,-82.168,-177.450,10.814,149.508
C06894=1115.247,335.301,-82.139,-177.453,10.812,149.509
C06895=1115.251,335.088,-82.110,-177.456,10.809,149.509
C06896=1115.254,334.876,-82.080,-177.459,10.808,149.509
C06897=1115.258,334.664,-82.051,-177.461,10.806,149.509
C06898=1115.261,334.452,-82.022,-177.464,10.803,149.509
C06899=1115.264,334.239,-81.993,-177.467,10.801,149.509
C06900=1115.268,333.992,-81.959,-177.470,10.799,149.510
C06901=1115.272,333.744,-81.924,-177.473,10.796,149.510
C06902=1115.276,333.497,-81.890,-177.476,10.794,149.510
C06903=1115.280,333.248,-81.856,-177.479,10.791,149.510
C06904=1115.284,333.001,-81.822,-177.483,10.789,149.510
C06905=1115.288,332.754,-81.788,-177.486,10.786,149.511
C06906=1115.292,332.506,-81.753,-177.489,10.783,149.511
C06907=1115.296,332.258,-81.720,-177.492,10.782,149.511
C06908=1115.300,332.011,-81.686,-177.495,10.779,149.511
C06909=1115.304,331.763,-81.652,-177.498,10.777,149.511
C06910=1115.308,331.516,-81.618,-177.501,10.774,149.512
C06911=1115.311,331.267,-81.584,-177.505,10.772,149.512
C06912=1115.316,331.020,-81.550,-177.507,10.769,149.512
C06913=1115.320,330.772,-81.517,-177.511,10.766,149.512
C06914=1115.323,330.524,-81.482,-177.514,10.764,149.512
C06915=1115.327,330.277,-81.448,-177.517,10.762,149.513
C06916=1115.332,330.029,-81.415,-177.520,10.759,149.513
C06917=1115.336,329.782,-81.381,-177.524,10.756,149.513
C06918=1115.339,329.533,-81.347,-177.527,10.754,149.513
C06919=1115.343,329.286,-81.313,-177.529,10.752,149.513
C06920=1115.348,329.039,-81.279,-177.533,10.749,149.513
C06921=1115.351,328.791,-81.245,-177.536,10.747,149.514
C06922=1115.355,328.543,-81.212,-177.539,10.744,149.514
C06923=1115.359,328.296,-81.178,-177.542,10.742,149.514
C06924=1115.363,328.048,-81.144,-177.545,10.739,149.514
C06925=1115.367,327.800,-81.110,-177.548,10.736,149.514
C06926=1115.371,327.552,-81.077,-177.552,10.734,149.515
C06927=1115.375,327.305,-81.043,-177.555,10.732,149.515
C06928=1115.379,327.057,-81.010,-177.558,10.729,149.515
C06929=1115.383,326.809,-80.976,-177.561,10.726,149.515
C06930=1115.388,326.561,-80.942,-177.564,10.725,149.515
C06931=1115.392,326.314,-80.909,-177.567,10.722,149.515
C06932=1115.395,326.067,-80.875,-177.570,10.719,149.516
C06933=1115.399,325.818,-80.842,-177.574,10.717,149.516
C06934=1115.403,325.571,-80.808,-177.576,10.714,149.516
C06935=1115.407,325.323,-80.775,-177.580,10.712,149.516
C06936=1115.411,325.076,-80.742,-177.583,10.709,149.517
C06937=1115.415,324.827,-80.708,-177.586,10.707,149.517
C06938=1115.419,324.580,-80.674,-177.589,10.704,149.517
C06939=1115.423,324.332,-80.641,-177.593,10.702,149.517
C06940=1115.427,324.085,-80.608,-177.596,10.699,149.517
C06941=1115.431,323.837,-80.573,-177.598,10.697,149.517
C06942=1115.435,323.589,-80.540,-177.602,10.695,149.518
C06943=1115.439,323.341,-80.507,-177.605,10.692,149.518
C06944=1115.443,323.093,-80.474,-177.608,10.690,149.518
C06945=1115.447,322.846,-80.440,-177.611,10.687,149.518
C06946=1115.451,322.598,-80.406,-177.614,10.684,149.518
C06947=1115.455,322.351,-80.373,-177.617,10.682,149.519
C06948=1115.458,322.138,-80.345,-177.620,10.680,149.519
C06949=1115.462,321.925,-80.316,-177.623,10.677,149.519
C06950=1115.465,321.713,-80.288,-177.625,10.675,149.519
C06951=1115.468,321.501,-80.259,-177.628,10.674,149.519
C06952=1115.472,321.289,-80.231,-177.631,10.671,149.519
C06953=1115.475,321.076,-80.203,-177.633,10.669,149.519
C06954=1115.479,320.864,-80.175,-177.636,10.667,149.520
C06955=1115.482,320.651,-80.146,-177.639,10.665,149.520
C06956=1115.486,320.403,-80.113,-177.642,10.662,149.520
C06957=1115.491,320.156,-80.079,-177.645,10.659,149.520
C06958=1115.494,319.908,-80.047,-177.648,10.657,149.520
C06959=1115.498,319.660,-80.014,-177.651,10.655,149.521
C06960=1115.502,319.413,-79.981,-177.654,10.652,149.521
C06961=1115.506,319.164,-79.947,-177.657,10.650,149.521
C06962=1115.510,318.917,-79.914,-177.660,10.647,149.521
C06963=1115.514,318.669,-79.881,-177.664,10.645,149.521
C06964=1115.518,318.421,-79.848,-177.667,10.642,149.521
C06965=1115.522,318.174,-79.815,-177.670,10.640,149.522
C06966=1115.526,317.926,-79.782,-177.673,10.637,149.522
C06967=1115.530,317.678,-79.749,-177.677,10.635,149.522
C06968=1115.534,317.430,-79.716,-177.679,10.632,149.522
C06969=1115.538,317.183,-79.682,-177.683,10.629,149.522
C06970=1115.542,316.935,-79.651,-177.685,10.627,149.522
C06971=1115.546,316.687,-79.617,-177.688,10.625,149.523
C06972=1115.550,316.439,-79.584,-177.692,10.623,149.523
C06973=1115.554,316.192,-79.551,-177.695,10.620,149.523
C06974=1115.558,315.944,-79.518,-177.698,10.617,149.523
C06975=1115.562,315.696,-79.485,-177.701,10.615,149.523
C06976=1115.566,315.448,-79.453,-177.704,10.612,149.524
C06977=1115.570,315.200,-79.420,-177.708,10.610,149.524
C06978=1115.574,314.953,-79.387,-177.710,10.607,149.524
C06979=1115.578,314.705,-79.355,-177.714,10.605,149.524
C06980=1115.582,314.457,-79.322,-177.717,10.602,149.524
C06981=1115.587,314.209,-79.288,-177.719,10.600,149.525
C06982=1115.590,313.962,-79.256,-177.722,10.597,149.525
C06983=1115.594,313.713,-79.223,-177.726,10.595,149.525
C06984=1115.598,313.466,-79.190,-177.729,10.592,149.525
C06985=1115.602,313.218,-79.158,-177.732,10.590,149.525
C06986=1115.606,312.970,-79.125,-177.735,10.587,149.525
C06987=1115.610,312.722,-79.092,-177.738,10.584,149.526
C06988=1115.614,312.474,-79.060,-177.742,10.582,149.526
C06989=1115.618,312.226,-79.027,-177.744,10.579,149.526
C06990=1115.622,311.978,-78.995,-177.748,10.577,149.526
C06991=1115.626,311.731,-78.962,-177.751,10.574,149.526
C06992=1115.630,311.483,-78.929,-177.753,10.572,149.526
C06993=1115.634,311.235,-78.897,-177.757,10.570,149.527
C06994=1115.639,310.988,-78.864,-177.760,10.567,149.527
C06995=1115.642,310.740,-78.832,-177.763,10.565,149.527
C06996=1115.647,310.492,-78.799,-177.766,10.562,149.527
C06997=1115.651,310.244,-78.767,-177.769,10.560,149.527
C06998=1115.655,309.996,-78.735,-177.773,10.557,149.528
C06999=1115.659,309.748,-78.702,-177.775,10.554,149.528
C07000=1115.663,309.500,-78.670,-177.779,10.552,149.528
C07001=1115.667,309.252,-78.637,-177.782,10.549,149.528
C07002=1115.671,309.005,-78.605,-177.785,10.547,149.528
C07003=1115.675,308.756,-78.573,-177.787,10.545,149.528
C07004=1115.678,308.544,-78.545,-177.791,10.542,149.529
C07005=1115.682,308.331,-78.517,-177.793,10.540,149.529
C07006=1115.685,308.120,-78.490,-177.795,10.538,149.529
C07007=1115.689,307.906,-78.461,-177.799,10.536,149.529
C07008=1115.693,307.694,-78.434,-177.801,10.534,149.529
C07009=1115.696,307.482,-78.406,-177.803,10.532,149.529
C07010=1115.699,307.268,-78.379,-177.807,10.529,149.530
C07011=1115.703,307.057,-78.351,-177.809,10.527,149.530
C07012=1115.707,306.808,-78.318,-177.812,10.525,149.530
C07013=1115.711,306.560,-78.286,-177.815,10.522,149.530
C07014=1115.715,306.313,-78.255,-177.818,10.520,149.530
C07015=1115.719,306.065,-78.222,-177.821,10.517,149.530
C07016=1115.723,305.817,-78.190,-177.825,10.515,149.531
C07017=1115.727,305.569,-78.158,-177.828,10.512,149.531
C07018=1115.731,305.321,-78.126,-177.831,10.509,149.531
C07019=1115.736,305.073,-78.094,-177.833,10.507,149.531
C07020=1115.740,304.825,-78.062,-177.837,10.505,149.531
C07021=1115.743,304.578,-78.029,-177.840,10.502,149.531
C07022=1115.748,304.329,-77.997,-177.843,10.500,149.532
C07023=1115.752,304.082,-77.965,-177.846,10.497,149.532
C07024=1115.756,303.834,-77.933,-177.849,10.495,149.532
C07025=1115.760,303.586,-77.901,-177.852,10.492,149.532
C07026=1115.764,303.338,-77.869,-177.855,10.489,149.532
C07027=1115.768,303.090,-77.838,-177.858,10.487,149.532
C07028=1115.773,302.842,-77.805,-177.862,10.484,149.533
C07029=1115.776,302.594,-77.773,-177.864,10.482,149.533
C07030=1115.781,302.346,-77.742,-177.867,10.480,149.533
C07031=1115.785,302.098,-77.709,-177.870,10.477,149.533
C07032=1115.789,301.850,-77.678,-177.874,10.474,149.533
C07033=1115.793,301.603,-77.646,-177.876,10.472,149.533
C07034=1115.797,301.355,-77.614,-177.880,10.469,149.534
C07035=1115.801,301.106,-77.582,-177.883,10.467,149.534
C07036=1115.805,300.858,-77.550,-177.886,10.464,149.534
C07037=1115.809,300.611,-77.519,-177.889,10.462,149.534
C07038=1115.813,300.363,-77.487,-177.892,10.459,149.534
C07039=1115.817,300.115,-77.454,-177.895,10.457,149.535
C07040=1115.822,299.867,-77.423,-177.898,10.454,149.535
C07041=1115.826,299.619,-77.392,-177.901,10.452,149.535
C07042=1115.830,299.371,-77.360,-177.904,10.449,149.535
C07043=1115.834,299.123,-77.328,-177.907,10.446,149.535
C07044=1115.838,298.875,-77.296,-177.910,10.444,149.536
C07045=1115.843,298.628,-77.264,-177.913,10.441,149.536
C07046=1115.846,298.379,-77.233,-177.917,10.439,149.536
C07047=1115.850,298.131,-77.201,-177.920,10.436,149.536
C07048=1115.855,297.883,-77.170,-177.923,10.434,149.536
C07049=1115.858,297.635,-77.138,-177.925,10.432,149.536
C07050=1115.862,297.387,-77.106,-177.929,10.429,149.537
C07051=1115.867,297.139,-77.076,-177.932,10.426,149.537
C07052=1115.871,296.891,-77.043,-177.935,10.424,149.537
C07053=1115.875,296.644,-77.012,-177.938,10.421,149.537
C07054=1115.879,296.395,-76.980,-177.941,10.419,149.537
C07055=1115.884,296.148,-76.949,-177.944,10.416,149.537
C07056=1115.887,295.900,-76.917,-177.947,10.414,149.538
C07057=1115.891,295.651,-76.886,-177.950,10.411,149.538
C07058=1115.896,295.404,-76.855,-177.954,10.408,149.538
C07059=1115.899,295.156,-76.823,-177.956,10.406,149.538
C07060=1115.903,294.943,-76.796,-177.959,10.404,149.538
C07061=1115.907,294.730,-76.769,-177.962,10.402,149.538
C07062=1115.910,294.518,-76.742,-177.964,10.400,149.539
C07063=1115.914,294.305,-76.716,-177.967,10.397,149.539
C07064=1115.918,294.092,-76.689,-177.970,10.396,149.539
C07065=1115.920,293.879,-76.662,-177.972,10.394,149.539
C07066=1115.924,293.667,-76.634,-177.975,10.391,149.539
C07067=1115.928,293.454,-76.608,-177.977,10.389,149.539
C07068=1115.932,293.207,-76.577,-177.980,10.386,149.540
C07069=1115.936,292.958,-76.545,-177.983,10.384,149.540
C07070=1115.940,292.711,-76.514,-177.987,10.381,149.540
C07071=1115.944,292.462,-76.483,-177.990,10.379,149.540
C07072=1115.949,292.215,-76.451,-177.993,10.376,149.540
C07073=1115.953,291.966,-76.420,-177.996,10.373,149.540
C07074=1115.957,291.718,-76.390,-177.999,10.372,149.541
C07075=1115.960,291.470,-76.358,-178.002,10.369,149.541
C07076=1115.965,291.222,-76.327,-178.005,10.366,149.541
C07077=1115.969,290.974,-76.296,-178.008,10.364,149.541
C07078=1115.973,290.726,-76.265,-178.011,10.361,149.541
C07079=1115.977,290.478,-76.234,-178.014,10.359,149.541
C07080=1115.982,290.230,-76.202,-178.017,10.356,149.542
C07081=1115.985,289.982,-76.172,-178.020,10.353,149.542
C07082=1115.989,289.734,-76.141,-178.023,10.351,149.542
C07083=1115.993,289.486,-76.109,-178.026,10.349,149.542
C07084=1115.998,289.238,-76.078,-178.029,10.346,149.542
C07085=1116.002,288.990,-76.047,-178.032,10.343,149.542
C07086=1116.006,288.741,-76.016,-178.035,10.341,149.543
C07087=1116.010,288.494,-75.985,-178.038,10.338,149.543
C07088=1116.014,288.246,-75.954,-178.042,10.336,149.543
C07089=1116.019,287.998,-75.924,-178.044,10.333,149.543
C07090=1116.023,287.749,-75.892,-178.048,10.331,149.543
C07091=1116.026,287.501,-75.862,-178.051,10.328,149.543
C07092=1116.031,287.254,-75.831,-178.053,10.326,149.544
C07093=1116.035,287.005,-75.800,-178.056,10.323,149.544
C07094=1116.039,286.757,-75.769,-178.059,10.321,149.544
C07095=1116.043,286.510,-75.739,-178.063,10.318,149.544
C07096=1116.047,286.261,-75.708,-178.066,10.316,149.544
C07097=1116.052,286.013,-75.677,-178.069,10.313,149.545
C07098=1116.056,285.764,-75.646,-178.072,10.310,149.545
C07099=1116.060,285.517,-75.616,-178.075,10.308,149.545
C07100=1116.064,285.270,-75.584,-178.078,10.305,149.545
C07101=1116.068,285.021,-75.553,-178.080,10.303,149.545
C07102=1116.072,284.773,-75.523,-178.084,10.301,149.545
C07103=1116.077,284.525,-75.492,-178.087,10.298,149.546
C07104=1116.081,284.277,-75.461,-178.090,10.296,149.546
C07105=1116.084,284.029,-75.431,-178.093,10.293,149.546
C07106=1116.089,283.781,-75.400,-178.096,10.290,149.546
C07107=1116.092,283.533,-75.369,-178.099,10.288,149.546
C07108=1116.097,283.284,-75.339,-178.102,10.285,149.546
C07109=1116.102,283.036,-75.309,-178.106,10.282,149.547
C07110=1116.106,282.788,-75.278,-178.108,10.280,149.547
C07111=1116.110,282.540,-75.247,-178.111,10.278,149.547
C07112=1116.114,282.292,-75.217,-178.114,10.275,149.547
C07113=1116.118,282.044,-75.186,-178.117,10.272,149.547
C07114=1116.122,281.796,-75.155,-178.120,10.270,149.548
C07115=1116.126,281.548,-75.125,-178.123,10.267,149.548
C07116=1116.130,281.335,-75.099,-178.126,10.266,149.548
C07117=1116.133,281.122,-75.073,-178.129,10.263,149.548
C07118=1116.137,280.910,-75.047,-178.131,10.261,149.548
C07119=1116.141,280.697,-75.021,-178.134,10.258,149.548
C07120=1116.145,280.484,-74.995,-178.137,10.257,149.549
C07121=1116.148,280.271,-74.969,-178.140,10.254,149.549
C07122=1116.152,280.058,-74.942,-178.142,10.252,149.549
C07123=1116.155,279.845,-74.916,-178.145,10.249,149.549
C07124=1116.160,279.597,-74.886,-178.148,10.247,149.549
C07125=1116.164,279.349,-74.856,-178.151,10.244,149.549
C07126=1116.168,279.100,-74.825,-178.155,10.241,149.550
C07127=1116.172,278.853,-74.795,-178.158,10.239,149.550
C07128=1116.176,278.604,-74.766,-178.161,10.236,149.550
C07129=1116.180,278.357,-74.735,-178.164,10.233,149.550
C07130=1116.184,278.109,-74.705,-178.167,10.231,149.550
C07131=1116.189,277.860,-74.674,-178.170,10.228,149.550
C07132=1116.193,277.612,-74.644,-178.173,10.226,149.550
C07133=1116.196,277.364,-74.614,-178.176,10.223,149.551
C07134=1116.201,277.116,-74.584,-178.179,10.220,149.551
C07135=1116.205,276.868,-74.554,-178.182,10.218,149.551
C07136=1116.210,276.620,-74.524,-178.185,10.215,149.551
C07137=1116.213,276.371,-74.493,-178.188,10.212,149.551
C07138=1116.218,276.123,-74.464,-178.191,10.209,149.551
C07139=1116.222,275.875,-74.433,-178.194,10.207,149.551
C07140=1116.226,275.627,-74.403,-178.198,10.204,149.552
C07141=1116.230,275.379,-74.373,-178.200,10.201,149.552
C07142=1116.235,275.131,-74.342,-178.203,10.199,149.552
C07143=1116.239,274.883,-74.313,-178.206,10.196,149.552
C07144=1116.243,274.634,-74.283,-178.209,10.193,149.552
C07145=1116.247,274.386,-74.253,-178.212,10.190,149.552
C07146=1116.251,274.138,-74.223,-178.216,10.188,149.552
C07147=1116.255,273.890,-74.193,-178.218,10.186,149.553
C07148=1116.260,273.642,-74.163,-178.221,10.183,149.553
C07149=1116.263,273.394,-74.133,-178.224,10.180,149.553
C07150=1116.268,273.145,-74.103,-178.227,10.178,149.553
C07151=1116.272,272.897,-74.074,-178.230,10.175,149.553
C07152=1116.276,272.650,-74.043,-178.233,10.172,149.553
C07153=1116.281,272.401,-74.014,-178.235,10.169,149.553
C07154=1116.285,272.153,-73.984,-178.238,10.167,149.553
C07155=1116.289,271.905,-73.954,-178.241,10.165,149.553
C07156=1116.293,271.656,-73.924,-178.244,10.162,149.554
C07157=1116.297,271.408,-73.895,-178.247,10.159,149.554
C07158=1116.301,271.160,-73.865,-178.250,10.157,149.554
C07159=1116.306,270.912,-73.834,-178.253,10.154,149.554
C07160=1116.310,270.663,-73.805,-178.256,10.151,149.554
C07161=1116.314,270.415,-73.775,-178.258,10.149,149.554
C07162=1116.318,270.167,-73.746,-178.261,10.146,149.554
C07163=1116.322,269.919,-73.716,-178.264,10.144,149.554
C07164=1116.326,269.671,-73.686,-178.267,10.141,149.554
C07165=1116.331,269.423,-73.657,-178.269,10.139,149.555
C07166=1116.336,269.174,-73.627,-178.272,10.136,149.555
C07167=1116.340,268.926,-73.597,-178.275,10.133,149.555
C07168=1116.344,268.677,-73.568,-178.278,10.131,149.555
C07169=1116.348,268.429,-73.538,-178.280,10.129,149.555
C07170=1116.352,268.182,-73.508,-178.283,10.126,149.555
C07171=1116.356,267.933,-73.479,-178.286,10.123,149.555
C07172=1116.360,267.721,-73.454,-178.289,10.121,149.555
C07173=1116.364,267.507,-73.429,-178.291,10.119,149.555
C07174=1116.367,267.294,-73.403,-178.293,10.117,149.555
C07175=1116.371,267.082,-73.378,-178.296,10.114,149.555
C07176=1116.375,266.869,-73.352,-178.298,10.112,149.556
C07177=1116.378,266.655,-73.327,-178.300,10.110,149.556
C07178=1116.382,266.443,-73.302,-178.303,10.108,149.556
C07179=1116.386,266.230,-73.276,-178.305,10.106,149.556
C07180=1116.390,265.982,-73.247,-178.308,10.103,149.556
C07181=1116.394,265.733,-73.218,-178.310,10.101,149.556
C07182=1116.398,265.485,-73.189,-178.313,10.099,149.556
C07183=1116.403,265.236,-73.159,-178.316,10.096,149.556
C07184=1116.407,264.988,-73.130,-178.318,10.094,149.557
C07185=1116.411,264.740,-73.100,-178.321,10.091,149.557
C07186=1116.416,264.492,-73.071,-178.324,10.089,149.557
C07187=1116.420,264.244,-73.042,-178.327,10.086,149.557
C07188=1116.424,263.996,-73.012,-178.331,10.083,149.557
C07189=1116.428,263.747,-72.983,-178.333,10.081,149.557
C07190=1116.432,263.499,-72.954,-178.336,10.078,149.557
C07191=1116.436,263.251,-72.925,-178.340,10.075,149.558
C07192=1116.440,263.002,-72.896,-178.343,10.072,149.558
C07193=1116.445,262.755,-72.867,-178.346,10.069,149.558
C07194=1116.449,262.506,-72.837,-178.350,10.067,149.558
C07195=1116.454,262.258,-72.808,-178.353,10.064,149.558
C07196=1116.458,262.010,-72.778,-178.356,10.060,149.558
C07197=1116.462,261.761,-72.750,-178.359,10.058,149.558
C07198=1116.466,261.513,-72.720,-178.362,10.055,149.559
C07199=1116.470,261.265,-72.691,-178.365,10.052,149.559
C07200=1116.475,261.017,-72.663,-178.368,10.050,149.559
C07201=1116.479,260.768,-72.634,-178.371,10.047,149.559
C07202=1116.483,260.520,-72.604,-178.374,10.044,149.559
C07203=1116.487,260.272,-72.575,-178.378,10.041,149.559
C07204=1116.491,260.023,-72.546,-178.381,10.038,149.559
C07205=1116.496,259.776,-72.517,-178.384,10.035,149.559
C07206=1116.501,259.527,-72.489,-178.387,10.032,149.560
C07207=1116.505,259.279,-72.459,-178.390,10.030,149.560
C07208=1116.508,259.031,-72.430,-178.392,10.027,149.560
C07209=1116.513,258.782,-72.402,-178.395,10.024,149.560
C07210=1116.517,258.534,-72.373,-178.398,10.021,149.560
C07211=1116.522,258.285,-72.344,-178.401,10.018,149.560
C07212=1116.525,258.037,-72.315,-178.404,10.015,149.560
C07213=1116.530,257.788,-72.286,-178.407,10.013,149.560
C07214=1116.535,257.541,-72.257,-178.410,10.010,149.560
C07215=1116.538,257.292,-72.229,-178.412,10.007,149.560
C07216=1116.543,257.044,-72.199,-178.415,10.004,149.560
C07217=1116.547,256.795,-72.171,-178.418,10.001,149.560
C07218=1116.551,256.548,-72.142,-178.421,9.999,149.561
C07219=1116.556,256.299,-72.114,-178.424,9.996,149.561
C07220=1116.560,256.051,-72.084,-178.426,9.993,149.561
C07221=1116.564,255.803,-72.056,-178.428,9.991,149.560
C07222=1116.568,255.555,-72.027,-178.429,9.990,149.560
C07223=1116.573,255.306,-71.998,-178.430,9.988,149.560
C07224=1116.577,255.058,-71.970,-178.432,9.985,149.560
C07225=1116.581,254.809,-71.941,-178.433,9.984,149.560
C07226=1116.586,254.561,-71.912,-178.435,9.982,149.560
C07227=1116.589,254.313,-71.883,-178.437,9.979,149.560
C07228=1116.594,254.099,-71.859,-178.439,9.978,149.560
C07229=1116.597,253.887,-71.835,-178.441,9.976,149.560
C07230=1116.601,253.673,-71.810,-178.442,9.975,149.560
C07231=1116.605,253.461,-71.785,-178.444,9.972,149.560
C07232=1116.608,253.247,-71.761,-178.446,9.971,149.560
C07233=1116.612,253.034,-71.736,-178.448,9.969,149.561
C07234=1116.615,252.821,-71.712,-178.451,9.967,149.561
C07235=1116.619,252.608,-71.688,-178.453,9.965,149.561
C07236=1116.624,252.360,-71.658,-178.456,9.963,149.561
C07237=1116.627,252.111,-71.630,-178.458,9.961,149.561
C07238=1116.632,251.863,-71.602,-178.461,9.958,149.561
C07239=1116.636,251.615,-71.573,-178.465,9.955,149.562
C07240=1116.641,251.367,-71.544,-178.467,9.953,149.562
C07241=1116.645,251.118,-71.516,-178.471,9.950,149.562
C07242=1116.649,250.869,-71.488,-178.474,9.947,149.562
C07243=1116.654,250.621,-71.460,-178.478,9.944,149.562
C07244=1116.658,250.373,-71.430,-178.482,9.941,149.563
C07245=1116.662,250.125,-71.402,-178.485,9.938,149.563
C07246=1116.667,249.876,-71.374,-178.489,9.935,149.563
C07247=1116.670,249.628,-71.346,-178.493,9.932,149.563
C07248=1116.675,249.380,-71.318,-178.497,9.929,149.564
C07249=1116.679,249.131,-71.289,-178.501,9.925,149.564
C07250=1116.684,248.883,-71.261,-178.505,9.921,149.564
C07251=1116.688,248.634,-71.233,-178.509,9.917,149.564
C07252=1116.692,248.386,-71.204,-178.513,9.914,149.565
C07253=1116.696,248.138,-71.177,-178.518,9.910,149.565
C07254=1116.701,247.889,-71.148,-178.523,9.906,149.565
C07255=1116.705,247.641,-71.120,-178.527,9.902,149.565
C07256=1116.709,247.392,-71.092,-178.531,9.899,149.566
C07257=1116.714,247.144,-71.064,-178.532,9.896,149.565
C07258=1116.718,246.896,-71.035,-178.534,9.894,149.565
C07259=1116.722,246.648,-71.008,-178.537,9.891,149.565
C07260=1116.726,246.399,-70.979,-178.539,9.888,149.565
C07261=1116.731,246.151,-70.951,-178.541,9.886,149.565
C07262=1116.734,245.902,-70.923,-178.543,9.884,149.565
C07263=1116.740,245.654,-70.895,-178.544,9.881,149.565
C07264=1116.744,245.405,-70.867,-178.547,9.878,149.565
C07265=1116.748,245.157,-70.839,-178.549,9.876,149.565
C07266=1116.752,244.908,-70.811,-178.551,9.874,149.565
C07267=1116.757,244.660,-70.783,-178.554,9.871,149.565
C07268=1116.761,244.412,-70.755,-178.556,9.869,149.565
C07269=1116.765,244.164,-70.727,-178.557,9.866,149.565
C07270=1116.770,243.914,-70.699,-178.559,9.864,149.565
C07271=1116.774,243.667,-70.671,-178.562,9.861,149.565
C07272=1116.778,243.419,-70.643,-178.564,9.859,149.565
C07273=1116.782,243.170,-70.615,-178.566,9.856,149.565
C07274=1116.787,242.922,-70.588,-178.569,9.854,149.565
C07275=1116.791,242.673,-70.560,-178.571,9.851,149.565
C07276=1116.796,242.425,-70.532,-178.573,9.848,149.565
C07277=1116.799,242.176,-70.504,-178.576,9.846,149.565
C07278=1116.804,241.928,-70.477,-178.578,9.844,149.565
C07279=1116.808,241.680,-70.449,-178.581,9.841,149.565
C07280=1116.812,241.431,-70.421,-178.583,9.839,149.565
